gfCNCPoint5[6043] = {X 587.4990, Y 6.7049, Z -6.3333, A 0.000, B 0.000, C 0.000 }
gfCNCPoint5[6044] = {X 587.4271, Y 5.9692, Z -6.3333, A 0.000, B 0.000, C 0.000 }
gfCNCPoint5[6045] = {X 587.4270, Y 5.0000, Z -6.3333, A 0.000, B 0.000, C 0.000 }
gfCNCPoint5[6046] = {X 587.5313, Y 4.0743, Z -6.3333, A 0.000, B 0.000, C 0.000 }
gfCNCPoint5[6047] = {X 587.8389, Y 3.1950, Z -6.3333, A 0.000, B 0.000, C 0.000 }
gfCNCPoint5[6048] = {X 588.3345, Y 2.4063, Z -6.3333, A 0.000, B 0.000, C 0.000 }
gfCNCPoint5[6049] = {X 588.9932, Y 1.7476, Z -6.3333, A 0.000, B 0.000, C 0.000 }
gfCNCPoint5[6050] = {X 589.7820, Y 1.2520, Z -6.3333, A 0.000, B 0.000, C 0.000 }
gfCNCPoint5[6051] = {X 590.6613, Y 0.9443, Z -6.3333, A 0.000, B 0.000, C 0.000 }
gfCNCPoint5[6052] = {X 591.5870, Y 0.8400, Z -6.3333, A 0.000, B 0.000, C 0.000 }
gfCNCPoint5[6053] = {X 600.0000, Y 0.8400, Z -6.3333, A 0.000, B 0.000, C 0.000 }
gfCNCPoint5[6054] = {X 600.8245, Y 0.9225, Z -6.3333, A 0.000, B 0.000, C 0.000 }
gfCNCPoint5[6055] = {X 601.6162, Y 1.1668, Z -6.3333, A 0.000, B 0.000, C 0.000 }
gfCNCPoint5[6056] = {X 602.3439, Y 1.5632, Z -6.3333, A 0.000, B 0.000, C 0.000 }
gfCNCPoint5[6057] = {X 602.9785, Y 2.0959, Z -6.3333, A 0.000, B 0.000, C 0.000 }
gfCNCPoint5[6058] = {X 603.4950, Y 2.7438, Z -6.3333, A 0.000, B 0.000, C 0.000 }
gfCNCPoint5[6059] = {X 603.6000, Y 2.9154, Z -6.3333, A 0.000, B 0.000, C 0.000 }
gfCNCPoint5[6060] = {X 603.6966, Y 3.0920, Z -6.3333, A 0.000, B 0.000, C 0.000 }
gfCNCPoint5[6061] = {X 607.6966, Y 10.8417, Z -6.3333, A 0.000, B 0.000, C 0.000 }
gfCNCPoint5[6062] = {X 607.6966, Y 10.8417, Z -3.3333, A 0.000, B 0.000, C 0.000 }
gfCNCPoint5[6063] = {X 607.6966, Y 10.8417, Z 11.0000, A 0.000, B 0.000, C 0.000 }
gfCNCPoint5[6064] = {X 607.6966, Y 38.1629, Z 11.0000, A 0.000, B 0.000, C 0.000 }
gfCNCPoint5[6065] = {X 607.6966, Y 38.1629, Z -3.3333, A 0.000, B 0.000, C 0.000 }
gfCNCPoint5[6066] = {X 607.6966, Y 38.1629, Z -6.3333, A 0.000, B 0.000, C 0.000 }
gfCNCPoint5[6067] = {X 603.6966, Y 46.7266, Z -6.3333, A 0.000, B 0.000, C 0.000 }
gfCNCPoint5[6068] = {X 603.5705, Y 46.9743, Z -6.3333, A 0.000, B 0.000, C 0.000 }
gfCNCPoint5[6069] = {X 603.4278, Y 47.2128, Z -6.3333, A 0.000, B 0.000, C 0.000 }
gfCNCPoint5[6070] = {X 602.9212, Y 47.8483, Z -6.3333, A 0.000, B 0.000, C 0.000 }
gfCNCPoint5[6071] = {X 602.2988, Y 48.3708, Z -6.3333, A 0.000, B 0.000, C 0.000 }
gfCNCPoint5[6072] = {X 601.5851, Y 48.7595, Z -6.3333, A 0.000, B 0.000, C 0.000 }
gfCNCPoint5[6073] = {X 600.8086, Y 48.9991, Z -6.3333, A 0.000, B 0.000, C 0.000 }
gfCNCPoint5[6074] = {X 600.0000, Y 49.0800, Z -6.3333, A 0.000, B 0.000, C 0.000 }
gfCNCPoint5[6075] = {X 593.5565, Y 49.0800, Z -6.3333, A 0.000, B 0.000, C 0.000 }
gfCNCPoint5[6076] = {X 592.6486, Y 48.9777, Z -6.3333, A 0.000, B 0.000, C 0.000 }
gfCNCPoint5[6077] = {X 591.7863, Y 48.6760, Z -6.3333, A 0.000, B 0.000, C 0.000 }
gfCNCPoint5[6078] = {X 591.0127, Y 48.1899, Z -6.3333, A 0.000, B 0.000, C 0.000 }
gfCNCPoint5[6079] = {X 590.3667, Y 47.5438, Z -6.3333, A 0.000, B 0.000, C 0.000 }
gfCNCPoint5[6080] = {X 589.8806, Y 46.7702, Z -6.3333, A 0.000, B 0.000, C 0.000 }
gfCNCPoint5[6081] = {X 589.5788, Y 45.9079, Z -6.3333, A 0.000, B 0.000, C 0.000 }
gfCNCPoint5[6082] = {X 589.4765, Y 45.0000, Z -6.3333, A 0.000, B 0.000, C 0.000 }
gfCNCPoint5[6083] = {X 589.4765, Y 44.0656, Z -6.3333, A 0.000, B 0.000, C 0.000 }
gfCNCPoint5[6084] = {X 589.5808, Y 43.1618, Z -6.3333, A 0.000, B 0.000, C 0.000 }
gfCNCPoint5[6085] = {X 589.8809, Y 42.3029, Z -6.3333, A 0.000, B 0.000, C 0.000 }
gfCNCPoint5[6086] = {X 590.3624, Y 41.5308, Z -6.3333, A 0.000, B 0.000, C 0.000 }
gfCNCPoint5[6087] = {X 591.0016, Y 40.8833, Z -6.3333, A 0.000, B 0.000, C 0.000 }
gfCNCPoint5[6088] = {X 591.0024, Y 32.3007, Z -6.3333, A 0.000, B 0.000, C 0.000 }
gfCNCPoint5[6089] = {X 585.2236, Y 46.5606, Z -6.3333, A 0.000, B 0.000, C 0.000 }
gfCNCPoint5[6090] = {X 584.8743, Y 47.2242, Z -6.3333, A 0.000, B 0.000, C 0.000 }
gfCNCPoint5[6091] = {X 584.4095, Y 47.8125, Z -6.3333, A 0.000, B 0.000, C 0.000 }
gfCNCPoint5[6092] = {X 583.8449, Y 48.3059, Z -6.3333, A 0.000, B 0.000, C 0.000 }
gfCNCPoint5[6093] = {X 583.1996, Y 48.6877, Z -6.3333, A 0.000, B 0.000, C 0.000 }
gfCNCPoint5[6094] = {X 582.3082, Y 48.9895, Z -6.3333, A 0.000, B 0.000, C 0.000 }
gfCNCPoint5[6095] = {X 581.3715, Y 49.0792, Z -6.3333, A 0.000, B 0.000, C 0.000 }
gfCNCPoint5[6096] = {X 580.4391, Y 48.9518, Z -6.3333, A 0.000, B 0.000, C 0.000 }
gfCNCPoint5[6097] = {X 579.5607, Y 48.6142, Z -6.3333, A 0.000, B 0.000, C 0.000 }
gfCNCPoint5[6098] = {X 578.7830, Y 48.0843, Z -6.3333, A 0.000, B 0.000, C 0.000 }
gfCNCPoint5[6099] = {X 578.1474, Y 47.3903, Z -6.3333, A 0.000, B 0.000, C 0.000 }
gfCNCPoint5[6100] = {X 577.6877, Y 46.5692, Z -6.3333, A 0.000, B 0.000, C 0.000 }
gfCNCPoint5[6101] = {X 571.7795, Y 32.1221, Z -6.3333, A 0.000, B 0.000, C 0.000 }
gfCNCPoint5[6102] = {X 571.7798, Y 40.8840, Z -6.3333, A 0.000, B 0.000, C 0.000 }
gfCNCPoint5[6103] = {X 571.8686, Y 40.9570, Z -6.3333, A 0.000, B 0.000, C 0.000 }
gfCNCPoint5[6104] = {X 572.4697, Y 41.5905, Z -6.3333, A 0.000, B 0.000, C 0.000 }
gfCNCPoint5[6105] = {X 572.9222, Y 42.3373, Z -6.3333, A 0.000, B 0.000, C 0.000 }
gfCNCPoint5[6106] = {X 573.2054, Y 43.1634, Z -6.3333, A 0.000, B 0.000, C 0.000 }
gfCNCPoint5[6107] = {X 573.3063, Y 44.0308, Z -6.3333, A 0.000, B 0.000, C 0.000 }
gfCNCPoint5[6108] = {X 573.3064, Y 45.0000, Z -6.3333, A 0.000, B 0.000, C 0.000 }
gfCNCPoint5[6109] = {X 573.2041, Y 45.9079, Z -6.3333, A 0.000, B 0.000, C 0.000 }
gfCNCPoint5[6110] = {X 572.9024, Y 46.7702, Z -6.3333, A 0.000, B 0.000, C 0.000 }
gfCNCPoint5[6111] = {X 572.4163, Y 47.5438, Z -6.3333, A 0.000, B 0.000, C 0.000 }
gfCNCPoint5[6112] = {X 571.7703, Y 48.1899, Z -6.3333, A 0.000, B 0.000, C 0.000 }
gfCNCPoint5[6113] = {X 570.9967, Y 48.6760, Z -6.3333, A 0.000, B 0.000, C 0.000 }
gfCNCPoint5[6114] = {X 570.1343, Y 48.9777, Z -6.3333, A 0.000, B 0.000, C 0.000 }
gfCNCPoint5[6115] = {X 569.2264, Y 49.0800, Z -6.3333, A 0.000, B 0.000, C 0.000 }
gfCNCPoint5[6116] = {X 562.4443, Y 49.0800, Z -6.3333, A 0.000, B 0.000, C 0.000 }
gfCNCPoint5[6117] = {X 561.5364, Y 48.9777, Z -6.3333, A 0.000, B 0.000, C 0.000 }
gfCNCPoint5[6118] = {X 560.6741, Y 48.6760, Z -6.3333, A 0.000, B 0.000, C 0.000 }
gfCNCPoint5[6119] = {X 559.9005, Y 48.1899, Z -6.3333, A 0.000, B 0.000, C 0.000 }
gfCNCPoint5[6120] = {X 559.2544, Y 47.5438, Z -6.3333, A 0.000, B 0.000, C 0.000 }
gfCNCPoint5[6121] = {X 558.7683, Y 46.7702, Z -6.3333, A 0.000, B 0.000, C 0.000 }
gfCNCPoint5[6122] = {X 558.4666, Y 45.9079, Z -6.3333, A 0.000, B 0.000, C 0.000 }
gfCNCPoint5[6123] = {X 558.3643, Y 45.0000, Z -6.3333, A 0.000, B 0.000, C 0.000 }
gfCNCPoint5[6124] = {X 558.3643, Y 44.0657, Z -6.3333, A 0.000, B 0.000, C 0.000 }
gfCNCPoint5[6125] = {X 558.4683, Y 43.1614, Z -6.3333, A 0.000, B 0.000, C 0.000 }
gfCNCPoint5[6126] = {X 558.7688, Y 42.3022, Z -6.3333, A 0.000, B 0.000, C 0.000 }
gfCNCPoint5[6127] = {X 559.2510, Y 41.5302, Z -6.3333, A 0.000, B 0.000, C 0.000 }
gfCNCPoint5[6128] = {X 559.8912, Y 40.8832, Z -6.3333, A 0.000, B 0.000, C 0.000 }
gfCNCPoint5[6129] = {X 559.8912, Y 9.1165, Z -6.3333, A 0.000, B 0.000, C 0.000 }
gfCNCPoint5[6130] = {X 559.2544, Y 8.4779, Z -6.3333, A 0.000, B 0.000, C 0.000 }
gfCNCPoint5[6131] = {X 558.7735, Y 7.7150, Z -6.3333, A 0.000, B 0.000, C 0.000 }
gfCNCPoint5[6132] = {X 558.4720, Y 6.8651, Z -6.3333, A 0.000, B 0.000, C 0.000 }
gfCNCPoint5[6133] = {X 558.3645, Y 5.9697, Z -6.3333, A 0.000, B 0.000, C 0.000 }
gfCNCPoint5[6134] = {X 558.3643, Y 5.0000, Z -6.3333, A 0.000, B 0.000, C 0.000 }
gfCNCPoint5[6135] = {X 558.4666, Y 4.0921, Z -6.3333, A 0.000, B 0.000, C 0.000 }
gfCNCPoint5[6136] = {X 558.7683, Y 3.2298, Z -6.3333, A 0.000, B 0.000, C 0.000 }
gfCNCPoint5[6137] = {X 559.2544, Y 2.4562, Z -6.3333, A 0.000, B 0.000, C 0.000 }
gfCNCPoint5[6138] = {X 559.9005, Y 1.8101, Z -6.3333, A 0.000, B 0.000, C 0.000 }
gfCNCPoint5[6139] = {X 560.6741, Y 1.3240, Z -6.3333, A 0.000, B 0.000, C 0.000 }
gfCNCPoint5[6140] = {X 561.5364, Y 1.0223, Z -6.3333, A 0.000, B 0.000, C 0.000 }
gfCNCPoint5[6141] = {X 562.4443, Y 0.9200, Z -6.3333, A 0.000, B 0.000, C 0.000 }
gfCNCPoint5[6142] = {X 570.9376, Y 0.9200, Z -6.3333, A 0.000, B 0.000, C 0.000 }
gfCNCPoint5[6143] = {X 571.8454, Y 1.0223, Z -6.3333, A 0.000, B 0.000, C 0.000 }
gfCNCPoint5[6144] = {X 572.7078, Y 1.3240, Z -6.3333, A 0.000, B 0.000, C 0.000 }
gfCNCPoint5[6145] = {X 573.4814, Y 1.8101, Z -6.3333, A 0.000, B 0.000, C 0.000 }
gfCNCPoint5[6146] = {X 574.1274, Y 2.4562, Z -6.3333, A 0.000, B 0.000, C 0.000 }
gfCNCPoint5[6147] = {X 574.6135, Y 3.2298, Z -6.3333, A 0.000, B 0.000, C 0.000 }
gfCNCPoint5[6148] = {X 574.9153, Y 4.0921, Z -6.3333, A 0.000, B 0.000, C 0.000 }
gfCNCPoint5[6149] = {X 575.0176, Y 5.0000, Z -6.3333, A 0.000, B 0.000, C 0.000 }
gfCNCPoint5[6150] = {X 575.0176, Y 5.9342, Z -6.3333, A 0.000, B 0.000, C 0.000 }
gfCNCPoint5[6151] = {X 574.9500, Y 6.6733, Z -6.3333, A 0.000, B 0.000, C 0.000 }
gfCNCPoint5[6152] = {X 574.7497, Y 7.3880, Z -6.3333, A 0.000, B 0.000, C 0.000 }
gfCNCPoint5[6153] = {X 574.4233, Y 8.0545, Z -6.3333, A 0.000, B 0.000, C 0.000 }
gfCNCPoint5[6154] = {X 574.3788, Y 8.1258, Z -6.3333, A 0.000, B 0.000, C 0.000 }
gfCNCPoint5[6155] = {X 574.3330, Y 8.1963, Z -6.3333, A 0.000, B 0.000, C 0.000 }
gfCNCPoint5[6156] = {X 574.3593, Y 8.2418, Z -6.3333, A 0.000, B 0.000, C 0.000 }
gfCNCPoint5[6157] = {X 581.1906, Y 25.0042, Z -6.3333, A 0.000, B 0.000, C 0.000 }
gfCNCPoint5[6158] = {X 588.1131, Y 8.0738, Z -6.3333, A 0.000, B 0.000, C 0.000 }
gfCNCPoint5[6159] = {X 587.7843, Y 7.4127, Z -6.3333, A 0.000, B 0.000, C 0.000 }
gfCNCPoint5[6160] = {X 587.5801, Y 6.7032, Z -6.3333, A 0.000, B 0.000, C 0.000 }
gfCNCPoint5[6161] = {X 587.5071, Y 5.9685, Z -6.3333, A 0.000, B 0.000, C 0.000 }
gfCNCPoint5[6162] = {X 587.5070, Y 5.0000, Z -6.3333, A 0.000, B 0.000, C 0.000 }
gfCNCPoint5[6163] = {X 587.6092, Y 4.0921, Z -6.3333, A 0.000, B 0.000, C 0.000 }
gfCNCPoint5[6164] = {X 587.9110, Y 3.2298, Z -6.3333, A 0.000, B 0.000, C 0.000 }
gfCNCPoint5[6165] = {X 588.3971, Y 2.4562, Z -6.3333, A 0.000, B 0.000, C 0.000 }
gfCNCPoint5[6166] = {X 589.0431, Y 1.8101, Z -6.3333, A 0.000, B 0.000, C 0.000 }
gfCNCPoint5[6167] = {X 589.8167, Y 1.3240, Z -6.3333, A 0.000, B 0.000, C 0.000 }
gfCNCPoint5[6168] = {X 590.6791, Y 1.0223, Z -6.3333, A 0.000, B 0.000, C 0.000 }
gfCNCPoint5[6169] = {X 591.5870, Y 0.9200, Z -6.3333, A 0.000, B 0.000, C 0.000 }
gfCNCPoint5[6170] = {X 600.0000, Y 0.9200, Z -6.3333, A 0.000, B 0.000, C 0.000 }
gfCNCPoint5[6171] = {X 600.8086, Y 1.0009, Z -6.3333, A 0.000, B 0.000, C 0.000 }
gfCNCPoint5[6172] = {X 601.5851, Y 1.2405, Z -6.3333, A 0.000, B 0.000, C 0.000 }
gfCNCPoint5[6173] = {X 602.2988, Y 1.6292, Z -6.3333, A 0.000, B 0.000, C 0.000 }
gfCNCPoint5[6174] = {X 602.9212, Y 2.1517, Z -6.3333, A 0.000, B 0.000, C 0.000 }
gfCNCPoint5[6175] = {X 603.4278, Y 2.7872, Z -6.3333, A 0.000, B 0.000, C 0.000 }
gfCNCPoint5[6176] = {X 603.5705, Y 3.0257, Z -6.3333, A 0.000, B 0.000, C 0.000 }
gfCNCPoint5[6177] = {X 603.6966, Y 3.2734, Z -6.3333, A 0.000, B 0.000, C 0.000 }
gfCNCPoint5[6178] = {X 607.6966, Y 11.8371, Z -6.3333, A 0.000, B 0.000, C 0.000 }
gfCNCPoint5[6179] = {X 607.6966, Y 11.8371, Z -3.3333, A 0.000, B 0.000, C 0.000 }
gfCNCPoint5[6180] = {X 607.6966, Y 11.8371, Z 11.0000, A 0.000, B 0.000, C 0.000 }
gfCNCPoint5[6181] = {X 607.6966, Y 36.8512, Z 11.0000, A 0.000, B 0.000, C 0.000 }
gfCNCPoint5[6182] = {X 607.6966, Y 36.8512, Z -3.3333, A 0.000, B 0.000, C 0.000 }
gfCNCPoint5[6183] = {X 607.6966, Y 36.8512, Z -6.3333, A 0.000, B 0.000, C 0.000 }
gfCNCPoint5[6184] = {X 603.6966, Y 46.5280, Z -6.3333, A 0.000, B 0.000, C 0.000 }
gfCNCPoint5[6185] = {X 603.5432, Y 46.8564, Z -6.3333, A 0.000, B 0.000, C 0.000 }
gfCNCPoint5[6186] = {X 603.3606, Y 47.1694, Z -6.3333, A 0.000, B 0.000, C 0.000 }
gfCNCPoint5[6187] = {X 602.8640, Y 47.7924, Z -6.3333, A 0.000, B 0.000, C 0.000 }
gfCNCPoint5[6188] = {X 602.2537, Y 48.3047, Z -6.3333, A 0.000, B 0.000, C 0.000 }
gfCNCPoint5[6189] = {X 601.5541, Y 48.6858, Z -6.3333, A 0.000, B 0.000, C 0.000 }
gfCNCPoint5[6190] = {X 600.7928, Y 48.9207, Z -6.3333, A 0.000, B 0.000, C 0.000 }
gfCNCPoint5[6191] = {X 600.0000, Y 49.0000, Z -6.3333, A 0.000, B 0.000, C 0.000 }
gfCNCPoint5[6192] = {X 593.5565, Y 49.0000, Z -6.3333, A 0.000, B 0.000, C 0.000 }
gfCNCPoint5[6193] = {X 592.6664, Y 48.8997, Z -6.3333, A 0.000, B 0.000, C 0.000 }
gfCNCPoint5[6194] = {X 591.8210, Y 48.6039, Z -6.3333, A 0.000, B 0.000, C 0.000 }
gfCNCPoint5[6195] = {X 591.0626, Y 48.1273, Z -6.3333, A 0.000, B 0.000, C 0.000 }
gfCNCPoint5[6196] = {X 590.4292, Y 47.4940, Z -6.3333, A 0.000, B 0.000, C 0.000 }
gfCNCPoint5[6197] = {X 589.9527, Y 46.7355, Z -6.3333, A 0.000, B 0.000, C 0.000 }
gfCNCPoint5[6198] = {X 589.6568, Y 45.8901, Z -6.3333, A 0.000, B 0.000, C 0.000 }
gfCNCPoint5[6199] = {X 589.5565, Y 45.0000, Z -6.3333, A 0.000, B 0.000, C 0.000 }
gfCNCPoint5[6200] = {X 589.5565, Y 44.0660, Z -6.3333, A 0.000, B 0.000, C 0.000 }
gfCNCPoint5[6201] = {X 589.6609, Y 43.1705, Z -6.3333, A 0.000, B 0.000, C 0.000 }
gfCNCPoint5[6202] = {X 589.9613, Y 42.3204, Z -6.3333, A 0.000, B 0.000, C 0.000 }
gfCNCPoint5[6203] = {X 590.4428, Y 41.5582, Z -6.3333, A 0.000, B 0.000, C 0.000 }
gfCNCPoint5[6204] = {X 591.0815, Y 40.9218, Z -6.3333, A 0.000, B 0.000, C 0.000 }
gfCNCPoint5[6205] = {X 591.0821, Y 40.7351, Z -6.3333, A 0.000, B 0.000, C 0.000 }
gfCNCPoint5[6206] = {X 591.0834, Y 40.3069, Z -6.3333, A 0.000, B 0.000, C 0.000 }
gfCNCPoint5[6207] = {X 591.0823, Y 32.0438, Z -6.3333, A 0.000, B 0.000, C 0.000 }
gfCNCPoint5[6208] = {X 590.9675, Y 32.1736, Z -6.3333, A 0.000, B 0.000, C 0.000 }
gfCNCPoint5[6209] = {X 590.3119, Y 33.7916, Z -6.3333, A 0.000, B 0.000, C 0.000 }
gfCNCPoint5[6210] = {X 585.1497, Y 46.5300, Z -6.3333, A 0.000, B 0.000, C 0.000 }
gfCNCPoint5[6211] = {X 584.8073, Y 47.1805, Z -6.3333, A 0.000, B 0.000, C 0.000 }
gfCNCPoint5[6212] = {X 584.3516, Y 47.7574, Z -6.3333, A 0.000, B 0.000, C 0.000 }
gfCNCPoint5[6213] = {X 583.7980, Y 48.2411, Z -6.3333, A 0.000, B 0.000, C 0.000 }
gfCNCPoint5[6214] = {X 583.1653, Y 48.6154, Z -6.3333, A 0.000, B 0.000, C 0.000 }
gfCNCPoint5[6215] = {X 582.2878, Y 48.9121, Z -6.3333, A 0.000, B 0.000, C 0.000 }
gfCNCPoint5[6216] = {X 581.3656, Y 48.9990, Z -6.3333, A 0.000, B 0.000, C 0.000 }
gfCNCPoint5[6217] = {X 580.4480, Y 48.8715, Z -6.3333, A 0.000, B 0.000, C 0.000 }
gfCNCPoint5[6218] = {X 579.5845, Y 48.5363, Z -6.3333, A 0.000, B 0.000, C 0.000 }
gfCNCPoint5[6219] = {X 578.8212, Y 48.0115, Z -6.3333, A 0.000, B 0.000, C 0.000 }
gfCNCPoint5[6220] = {X 578.1990, Y 47.3251, Z -6.3333, A 0.000, B 0.000, C 0.000 }
gfCNCPoint5[6221] = {X 577.7515, Y 46.5141, Z -6.3333, A 0.000, B 0.000, C 0.000 }
gfCNCPoint5[6222] = {X 571.6995, Y 31.7151, Z -6.3333, A 0.000, B 0.000, C 0.000 }
gfCNCPoint5[6223] = {X 571.6998, Y 40.9218, Z -6.3333, A 0.000, B 0.000, C 0.000 }
gfCNCPoint5[6224] = {X 571.8386, Y 41.0366, Z -6.3333, A 0.000, B 0.000, C 0.000 }
gfCNCPoint5[6225] = {X 572.4243, Y 41.6631, Z -6.3333, A 0.000, B 0.000, C 0.000 }
gfCNCPoint5[6226] = {X 572.8630, Y 42.3999, Z -6.3333, A 0.000, B 0.000, C 0.000 }
gfCNCPoint5[6227] = {X 573.1345, Y 43.2134, Z -6.3333, A 0.000, B 0.000, C 0.000 }
gfCNCPoint5[6228] = {X 573.2264, Y 44.0660, Z -6.3333, A 0.000, B 0.000, C 0.000 }
gfCNCPoint5[6229] = {X 573.2264, Y 45.0000, Z -6.3333, A 0.000, B 0.000, C 0.000 }
gfCNCPoint5[6230] = {X 573.1261, Y 45.8901, Z -6.3333, A 0.000, B 0.000, C 0.000 }
gfCNCPoint5[6231] = {X 572.8303, Y 46.7355, Z -6.3333, A 0.000, B 0.000, C 0.000 }
gfCNCPoint5[6232] = {X 572.3538, Y 47.4940, Z -6.3333, A 0.000, B 0.000, C 0.000 }
gfCNCPoint5[6233] = {X 571.7204, Y 48.1273, Z -6.3333, A 0.000, B 0.000, C 0.000 }
gfCNCPoint5[6234] = {X 570.9620, Y 48.6039, Z -6.3333, A 0.000, B 0.000, C 0.000 }
gfCNCPoint5[6235] = {X 570.1165, Y 48.8997, Z -6.3333, A 0.000, B 0.000, C 0.000 }
gfCNCPoint5[6236] = {X 569.2264, Y 49.0000, Z -6.3333, A 0.000, B 0.000, C 0.000 }
gfCNCPoint5[6237] = {X 562.4443, Y 49.0000, Z -6.3333, A 0.000, B 0.000, C 0.000 }
gfCNCPoint5[6238] = {X 561.5542, Y 48.8997, Z -6.3333, A 0.000, B 0.000, C 0.000 }
gfCNCPoint5[6239] = {X 560.7088, Y 48.6039, Z -6.3333, A 0.000, B 0.000, C 0.000 }
gfCNCPoint5[6240] = {X 559.9503, Y 48.1273, Z -6.3333, A 0.000, B 0.000, C 0.000 }
gfCNCPoint5[6241] = {X 559.3170, Y 47.4940, Z -6.3333, A 0.000, B 0.000, C 0.000 }
gfCNCPoint5[6242] = {X 558.8404, Y 46.7355, Z -6.3333, A 0.000, B 0.000, C 0.000 }
gfCNCPoint5[6243] = {X 558.5446, Y 45.8901, Z -6.3333, A 0.000, B 0.000, C 0.000 }
gfCNCPoint5[6244] = {X 558.4443, Y 45.0000, Z -6.3333, A 0.000, B 0.000, C 0.000 }
gfCNCPoint5[6245] = {X 558.4443, Y 44.0660, Z -6.3333, A 0.000, B 0.000, C 0.000 }
gfCNCPoint5[6246] = {X 558.5484, Y 43.1700, Z -6.3333, A 0.000, B 0.000, C 0.000 }
gfCNCPoint5[6247] = {X 558.8492, Y 42.3197, Z -6.3333, A 0.000, B 0.000, C 0.000 }
gfCNCPoint5[6248] = {X 559.3315, Y 41.5575, Z -6.3333, A 0.000, B 0.000, C 0.000 }
gfCNCPoint5[6249] = {X 559.9712, Y 40.9217, Z -6.3333, A 0.000, B 0.000, C 0.000 }
gfCNCPoint5[6250] = {X 559.9712, Y 9.0779, Z -6.3333, A 0.000, B 0.000, C 0.000 }
gfCNCPoint5[6251] = {X 559.3294, Y 8.4436, Z -6.3333, A 0.000, B 0.000, C 0.000 }
gfCNCPoint5[6252] = {X 558.8462, Y 7.6815, Z -6.3333, A 0.000, B 0.000, C 0.000 }
gfCNCPoint5[6253] = {X 558.5461, Y 6.8306, Z -6.3333, A 0.000, B 0.000, C 0.000 }
gfCNCPoint5[6254] = {X 558.4443, Y 5.9340, Z -6.3333, A 0.000, B 0.000, C 0.000 }
gfCNCPoint5[6255] = {X 558.4443, Y 5.0000, Z -6.3333, A 0.000, B 0.000, C 0.000 }
gfCNCPoint5[6256] = {X 558.5446, Y 4.1099, Z -6.3333, A 0.000, B 0.000, C 0.000 }
gfCNCPoint5[6257] = {X 558.8404, Y 3.2645, Z -6.3333, A 0.000, B 0.000, C 0.000 }
gfCNCPoint5[6258] = {X 559.3170, Y 2.5060, Z -6.3333, A 0.000, B 0.000, C 0.000 }
gfCNCPoint5[6259] = {X 559.9503, Y 1.8727, Z -6.3333, A 0.000, B 0.000, C 0.000 }
gfCNCPoint5[6260] = {X 560.7088, Y 1.3961, Z -6.3333, A 0.000, B 0.000, C 0.000 }
gfCNCPoint5[6261] = {X 561.5542, Y 1.1003, Z -6.3333, A 0.000, B 0.000, C 0.000 }
gfCNCPoint5[6262] = {X 562.4443, Y 1.0000, Z -6.3333, A 0.000, B 0.000, C 0.000 }
gfCNCPoint5[6263] = {X 570.9376, Y 1.0000, Z -6.3333, A 0.000, B 0.000, C 0.000 }
gfCNCPoint5[6264] = {X 571.8276, Y 1.1003, Z -6.3333, A 0.000, B 0.000, C 0.000 }
gfCNCPoint5[6265] = {X 572.6731, Y 1.3961, Z -6.3333, A 0.000, B 0.000, C 0.000 }
gfCNCPoint5[6266] = {X 573.4315, Y 1.8727, Z -6.3333, A 0.000, B 0.000, C 0.000 }
gfCNCPoint5[6267] = {X 574.0649, Y 2.5060, Z -6.3333, A 0.000, B 0.000, C 0.000 }
gfCNCPoint5[6268] = {X 574.5414, Y 3.2645, Z -6.3333, A 0.000, B 0.000, C 0.000 }
gfCNCPoint5[6269] = {X 574.8373, Y 4.1099, Z -6.3333, A 0.000, B 0.000, C 0.000 }
gfCNCPoint5[6270] = {X 574.9376, Y 5.0000, Z -6.3333, A 0.000, B 0.000, C 0.000 }
gfCNCPoint5[6271] = {X 574.9372, Y 5.9858, Z -6.3333, A 0.000, B 0.000, C 0.000 }
gfCNCPoint5[6272] = {X 574.8650, Y 6.6926, Z -6.3333, A 0.000, B 0.000, C 0.000 }
gfCNCPoint5[6273] = {X 574.6688, Y 7.3755, Z -6.3333, A 0.000, B 0.000, C 0.000 }
gfCNCPoint5[6274] = {X 574.3549, Y 8.0129, Z -6.3333, A 0.000, B 0.000, C 0.000 }
gfCNCPoint5[6275] = {X 574.2921, Y 8.1128, Z -6.3333, A 0.000, B 0.000, C 0.000 }
gfCNCPoint5[6276] = {X 574.2264, Y 8.2108, Z -6.3333, A 0.000, B 0.000, C 0.000 }
gfCNCPoint5[6277] = {X 574.2617, Y 8.2359, Z -6.3333, A 0.000, B 0.000, C 0.000 }
gfCNCPoint5[6278] = {X 574.2853, Y 8.2722, Z -6.3333, A 0.000, B 0.000, C 0.000 }
gfCNCPoint5[6279] = {X 574.9161, Y 9.8071, Z -6.3333, A 0.000, B 0.000, C 0.000 }
gfCNCPoint5[6280] = {X 581.1904, Y 25.2159, Z -6.3333, A 0.000, B 0.000, C 0.000 }
gfCNCPoint5[6281] = {X 588.2026, Y 8.0662, Z -6.3333, A 0.000, B 0.000, C 0.000 }
gfCNCPoint5[6282] = {X 587.8646, Y 7.3984, Z -6.3333, A 0.000, B 0.000, C 0.000 }
gfCNCPoint5[6283] = {X 587.6570, Y 6.6792, Z -6.3333, A 0.000, B 0.000, C 0.000 }
gfCNCPoint5[6284] = {X 587.5870, Y 5.9340, Z -6.3333, A 0.000, B 0.000, C 0.000 }
gfCNCPoint5[6285] = {X 587.5870, Y 5.0000, Z -6.3333, A 0.000, B 0.000, C 0.000 }
gfCNCPoint5[6286] = {X 587.6872, Y 4.1099, Z -6.3333, A 0.000, B 0.000, C 0.000 }
gfCNCPoint5[6287] = {X 587.9831, Y 3.2645, Z -6.3333, A 0.000, B 0.000, C 0.000 }
gfCNCPoint5[6288] = {X 588.4596, Y 2.5060, Z -6.3333, A 0.000, B 0.000, C 0.000 }
gfCNCPoint5[6289] = {X 589.0930, Y 1.8727, Z -6.3333, A 0.000, B 0.000, C 0.000 }
gfCNCPoint5[6290] = {X 589.8514, Y 1.3961, Z -6.3333, A 0.000, B 0.000, C 0.000 }
gfCNCPoint5[6291] = {X 590.6969, Y 1.1003, Z -6.3333, A 0.000, B 0.000, C 0.000 }
gfCNCPoint5[6292] = {X 591.5870, Y 1.0000, Z -6.3333, A 0.000, B 0.000, C 0.000 }
gfCNCPoint5[6293] = {X 600.0000, Y 1.0000, Z -6.3333, A 0.000, B 0.000, C 0.000 }
gfCNCPoint5[6294] = {X 600.7928, Y 1.0793, Z -6.3333, A 0.000, B 0.000, C 0.000 }
gfCNCPoint5[6295] = {X 601.5541, Y 1.3142, Z -6.3333, A 0.000, B 0.000, C 0.000 }
gfCNCPoint5[6296] = {X 602.2537, Y 1.6953, Z -6.3333, A 0.000, B 0.000, C 0.000 }
gfCNCPoint5[6297] = {X 602.8640, Y 2.2076, Z -6.3333, A 0.000, B 0.000, C 0.000 }
gfCNCPoint5[6298] = {X 603.3606, Y 2.8306, Z -6.3333, A 0.000, B 0.000, C 0.000 }
gfCNCPoint5[6299] = {X 603.5432, Y 3.1436, Z -6.3333, A 0.000, B 0.000, C 0.000 }
gfCNCPoint5[6300] = {X 603.6966, Y 3.4720, Z -6.3333, A 0.000, B 0.000, C 0.000 }
gfCNCPoint5[6301] = {X 607.6966, Y 13.1488, Z -6.3333, A 0.000, B 0.000, C 0.000 }
gfCNCPoint5[6302] = {X 607.6966, Y 13.1488, Z -3.3333, A 0.000, B 0.000, C 0.000 }
gfCNCPoint5[6303] = {X 607.6966, Y 13.1488, Z 11.0000, A 0.000, B 0.000, C 0.000 }
gfCNCPoint5[6304] = {X 256.2463, Y 19.7817, Z 11.0000, A 0.000, B 0.000, C 0.000 }
gfCNCPoint5[6305] = {X 256.2463, Y 19.7817, Z -2.5000, A 0.000, B 0.000, C 0.000 }
gfCNCPoint5[6306] = {X 251.5292, Y 19.7817, Z -3.7639, A 0.000, B 0.000, C 0.000 }
gfCNCPoint5[6307] = {X 250.8344, Y 19.7926, Z -3.9501, A 0.000, B 0.000, C 0.000 }
gfCNCPoint5[6308] = {X 250.1815, Y 19.7939, Z -4.1251, A 0.000, B 0.000, C 0.000 }
gfCNCPoint5[6309] = {X 249.4949, Y 19.8924, Z -4.3110, A 0.000, B 0.000, C 0.000 }
gfCNCPoint5[6310] = {X 248.8454, Y 20.0807, Z -4.4922, A 0.000, B 0.000, C 0.000 }
gfCNCPoint5[6311] = {X 248.7086, Y 20.1119, Z -4.5298, A 0.000, B 0.000, C 0.000 }
gfCNCPoint5[6312] = {X 248.6548, Y 20.1623, Z -4.5495, A 0.000, B 0.000, C 0.000 }
gfCNCPoint5[6313] = {X 248.6149, Y 20.2969, Z -4.5871, A 0.000, B 0.000, C 0.000 }
gfCNCPoint5[6314] = {X 248.4759, Y 20.7652, Z -4.7180, A 0.000, B 0.000, C 0.000 }
gfCNCPoint5[6315] = {X 248.4457, Y 21.8668, Z -5.0133, A 0.000, B 0.000, C 0.000 }
gfCNCPoint5[6316] = {X 248.5589, Y 22.3420, Z -5.1442, A 0.000, B 0.000, C 0.000 }
gfCNCPoint5[6317] = {X 248.8757, Y 22.4372, Z -5.2328, A 0.000, B 0.000, C 0.000 }
gfCNCPoint5[6318] = {X 250.4427, Y 22.5655, Z -5.6541, A 0.000, B 0.000, C 0.000 }
gfCNCPoint5[6319] = {X 251.6873, Y 22.5560, Z -5.9876, A 0.000, B 0.000, C 0.000 }
gfCNCPoint5[6320] = {X 252.9776, Y 22.5560, Z -6.3333, A 0.000, B 0.000, C 0.000 }
gfCNCPoint5[6321] = {X 257.4115, Y 22.5560, Z -6.3333, A 0.000, B 0.000, C 0.000 }
gfCNCPoint5[6322] = {X 257.4115, Y 19.7817, Z -6.3333, A 0.000, B 0.000, C 0.000 }
gfCNCPoint5[6323] = {X 251.5292, Y 19.7817, Z -6.3333, A 0.000, B 0.000, C 0.000 }
gfCNCPoint5[6324] = {X 250.8344, Y 19.7926, Z -6.3333, A 0.000, B 0.000, C 0.000 }
gfCNCPoint5[6325] = {X 249.8296, Y 19.8658, Z -6.3333, A 0.000, B 0.000, C 0.000 }
gfCNCPoint5[6326] = {X 248.8454, Y 20.0807, Z -6.3333, A 0.000, B 0.000, C 0.000 }
gfCNCPoint5[6327] = {X 248.7009, Y 20.1576, Z -6.3333, A 0.000, B 0.000, C 0.000 }
gfCNCPoint5[6328] = {X 248.6149, Y 20.2969, Z -6.3333, A 0.000, B 0.000, C 0.000 }
gfCNCPoint5[6329] = {X 248.4770, Y 20.9719, Z -6.3333, A 0.000, B 0.000, C 0.000 }
gfCNCPoint5[6330] = {X 248.4582, Y 21.6605, Z -6.3333, A 0.000, B 0.000, C 0.000 }
gfCNCPoint5[6331] = {X 248.5589, Y 22.3420, Z -6.3333, A 0.000, B 0.000, C 0.000 }
gfCNCPoint5[6332] = {X 248.8789, Y 22.4201, Z -6.3333, A 0.000, B 0.000, C 0.000 }
gfCNCPoint5[6333] = {X 249.2053, Y 22.4642, Z -6.3333, A 0.000, B 0.000, C 0.000 }
gfCNCPoint5[6334] = {X 250.4453, Y 22.5379, Z -6.3333, A 0.000, B 0.000, C 0.000 }
gfCNCPoint5[6335] = {X 251.6873, Y 22.5560, Z -6.3333, A 0.000, B 0.000, C 0.000 }
gfCNCPoint5[6336] = {X 252.9776, Y 22.5560, Z -6.3333, A 0.000, B 0.000, C 0.000 }
gfCNCPoint5[6337] = {X 248.9928, Y 22.2874, Z -6.3333, A 0.000, B 0.000, C 0.000 }
gfCNCPoint5[6338] = {X 252.9776, Y 22.6360, Z -6.3333, A 0.000, B 0.000, C 0.000 }
gfCNCPoint5[6339] = {X 257.4915, Y 22.6360, Z -6.3333, A 0.000, B 0.000, C 0.000 }
gfCNCPoint5[6340] = {X 257.4915, Y 19.7017, Z -6.3333, A 0.000, B 0.000, C 0.000 }
gfCNCPoint5[6341] = {X 251.5286, Y 19.7017, Z -6.3333, A 0.000, B 0.000, C 0.000 }
gfCNCPoint5[6342] = {X 250.8364, Y 19.7126, Z -6.3333, A 0.000, B 0.000, C 0.000 }
gfCNCPoint5[6343] = {X 249.8259, Y 19.7859, Z -6.3333, A 0.000, B 0.000, C 0.000 }
gfCNCPoint5[6344] = {X 248.8357, Y 20.0009, Z -6.3333, A 0.000, B 0.000, C 0.000 }
gfCNCPoint5[6345] = {X 248.6492, Y 20.0964, Z -6.3333, A 0.000, B 0.000, C 0.000 }
gfCNCPoint5[6346] = {X 248.5382, Y 20.2741, Z -6.3333, A 0.000, B 0.000, C 0.000 }
gfCNCPoint5[6347] = {X 248.3958, Y 20.9779, Z -6.3333, A 0.000, B 0.000, C 0.000 }
gfCNCPoint5[6348] = {X 248.3803, Y 21.6958, Z -6.3333, A 0.000, B 0.000, C 0.000 }
gfCNCPoint5[6349] = {X 248.4919, Y 22.4051, Z -6.3333, A 0.000, B 0.000, C 0.000 }
gfCNCPoint5[6350] = {X 248.8415, Y 22.4943, Z -6.3333, A 0.000, B 0.000, C 0.000 }
gfCNCPoint5[6351] = {X 249.1988, Y 22.5439, Z -6.3333, A 0.000, B 0.000, C 0.000 }
gfCNCPoint5[6352] = {X 250.4414, Y 22.6178, Z -6.3333, A 0.000, B 0.000, C 0.000 }
gfCNCPoint5[6353] = {X 251.6861, Y 22.6360, Z -6.3333, A 0.000, B 0.000, C 0.000 }
gfCNCPoint5[6354] = {X 252.9776, Y 22.6360, Z -6.3333, A 0.000, B 0.000, C 0.000 }
gfCNCPoint5[6355] = {X 256.9624, Y 22.2874, Z -6.3333, A 0.000, B 0.000, C 0.000 }
gfCNCPoint5[6356] = {X 248.9928, Y 22.3674, Z -6.3333, A 0.000, B 0.000, C 0.000 }
gfCNCPoint5[6357] = {X 252.9776, Y 22.7160, Z -6.3333, A 0.000, B 0.000, C 0.000 }
gfCNCPoint5[6358] = {X 257.5715, Y 22.7160, Z -6.3333, A 0.000, B 0.000, C 0.000 }
gfCNCPoint5[6359] = {X 257.5715, Y 19.6217, Z -6.3333, A 0.000, B 0.000, C 0.000 }
gfCNCPoint5[6360] = {X 251.5280, Y 19.6217, Z -6.3333, A 0.000, B 0.000, C 0.000 }
gfCNCPoint5[6361] = {X 250.8357, Y 19.6326, Z -6.3333, A 0.000, B 0.000, C 0.000 }
gfCNCPoint5[6362] = {X 249.8156, Y 19.7065, Z -6.3333, A 0.000, B 0.000, C 0.000 }
gfCNCPoint5[6363] = {X 248.8161, Y 19.9232, Z -6.3333, A 0.000, B 0.000, C 0.000 }
gfCNCPoint5[6364] = {X 248.5938, Y 20.0386, Z -6.3333, A 0.000, B 0.000, C 0.000 }
gfCNCPoint5[6365] = {X 248.4615, Y 20.2513, Z -6.3333, A 0.000, B 0.000, C 0.000 }
gfCNCPoint5[6366] = {X 248.3147, Y 20.9838, Z -6.3333, A 0.000, B 0.000, C 0.000 }
gfCNCPoint5[6367] = {X 248.3025, Y 21.7308, Z -6.3333, A 0.000, B 0.000, C 0.000 }
gfCNCPoint5[6368] = {X 248.4254, Y 22.4676, Z -6.3333, A 0.000, B 0.000, C 0.000 }
gfCNCPoint5[6369] = {X 248.8042, Y 22.5685, Z -6.3333, A 0.000, B 0.000, C 0.000 }
gfCNCPoint5[6370] = {X 249.1923, Y 22.6236, Z -6.3333, A 0.000, B 0.000, C 0.000 }
gfCNCPoint5[6371] = {X 250.4383, Y 22.6977, Z -6.3333, A 0.000, B 0.000, C 0.000 }
gfCNCPoint5[6372] = {X 251.6864, Y 22.7160, Z -6.3333, A 0.000, B 0.000, C 0.000 }
gfCNCPoint5[6373] = {X 252.9776, Y 22.7160, Z -6.3333, A 0.000, B 0.000, C 0.000 }
gfCNCPoint5[6374] = {X 256.9624, Y 22.3674, Z -6.3333, A 0.000, B 0.000, C 0.000 }
gfCNCPoint5[6375] = {X 248.9928, Y 22.4474, Z -6.3333, A 0.000, B 0.000, C 0.000 }
gfCNCPoint5[6376] = {X 252.9776, Y 22.7960, Z -6.3333, A 0.000, B 0.000, C 0.000 }
gfCNCPoint5[6377] = {X 257.6515, Y 22.7960, Z -6.3333, A 0.000, B 0.000, C 0.000 }
gfCNCPoint5[6378] = {X 257.6515, Y 19.5417, Z -6.3333, A 0.000, B 0.000, C 0.000 }
gfCNCPoint5[6379] = {X 251.5274, Y 19.5417, Z -6.3333, A 0.000, B 0.000, C 0.000 }
gfCNCPoint5[6380] = {X 250.8350, Y 19.5526, Z -6.3333, A 0.000, B 0.000, C 0.000 }
gfCNCPoint5[6381] = {X 249.8053, Y 19.6272, Z -6.3333, A 0.000, B 0.000, C 0.000 }
gfCNCPoint5[6382] = {X 248.7963, Y 19.8457, Z -6.3333, A 0.000, B 0.000, C 0.000 }
gfCNCPoint5[6383] = {X 248.5383, Y 19.9810, Z -6.3333, A 0.000, B 0.000, C 0.000 }
gfCNCPoint5[6384] = {X 248.3848, Y 20.2286, Z -6.3333, A 0.000, B 0.000, C 0.000 }
gfCNCPoint5[6385] = {X 248.2337, Y 20.9896, Z -6.3333, A 0.000, B 0.000, C 0.000 }
gfCNCPoint5[6386] = {X 248.2250, Y 21.7655, Z -6.3333, A 0.000, B 0.000, C 0.000 }
gfCNCPoint5[6387] = {X 248.3592, Y 22.5297, Z -6.3333, A 0.000, B 0.000, C 0.000 }
gfCNCPoint5[6388] = {X 248.7670, Y 22.6425, Z -6.3333, A 0.000, B 0.000, C 0.000 }
gfCNCPoint5[6389] = {X 249.1857, Y 22.7034, Z -6.3333, A 0.000, B 0.000, C 0.000 }
gfCNCPoint5[6390] = {X 250.4352, Y 22.7777, Z -6.3333, A 0.000, B 0.000, C 0.000 }
gfCNCPoint5[6391] = {X 251.6867, Y 22.7960, Z -6.3333, A 0.000, B 0.000, C 0.000 }
gfCNCPoint5[6392] = {X 252.9776, Y 22.7960, Z -6.3333, A 0.000, B 0.000, C 0.000 }
gfCNCPoint5[6393] = {X 256.9624, Y 22.4474, Z -6.3333, A 0.000, B 0.000, C 0.000 }
gfCNCPoint5[6394] = {X 248.9928, Y 22.5274, Z -6.3333, A 0.000, B 0.000, C 0.000 }
gfCNCPoint5[6395] = {X 252.9776, Y 22.8760, Z -6.3333, A 0.000, B 0.000, C 0.000 }
gfCNCPoint5[6396] = {X 257.7315, Y 22.8760, Z -6.3333, A 0.000, B 0.000, C 0.000 }
gfCNCPoint5[6397] = {X 257.7315, Y 19.4617, Z -6.3333, A 0.000, B 0.000, C 0.000 }
gfCNCPoint5[6398] = {X 251.5267, Y 19.4617, Z -6.3333, A 0.000, B 0.000, C 0.000 }
gfCNCPoint5[6399] = {X 250.8343, Y 19.4726, Z -6.3333, A 0.000, B 0.000, C 0.000 }
gfCNCPoint5[6400] = {X 249.7949, Y 19.5478, Z -6.3333, A 0.000, B 0.000, C 0.000 }
gfCNCPoint5[6401] = {X 248.7763, Y 19.7682, Z -6.3333, A 0.000, B 0.000, C 0.000 }
gfCNCPoint5[6402] = {X 248.4828, Y 19.9234, Z -6.3333, A 0.000, B 0.000, C 0.000 }
gfCNCPoint5[6403] = {X 248.3081, Y 20.2058, Z -6.3333, A 0.000, B 0.000, C 0.000 }
gfCNCPoint5[6404] = {X 248.1533, Y 20.9889, Z -6.3333, A 0.000, B 0.000, C 0.000 }
gfCNCPoint5[6405] = {X 248.1465, Y 21.7871, Z -6.3333, A 0.000, B 0.000, C 0.000 }
gfCNCPoint5[6406] = {X 248.2880, Y 22.5727, Z -6.3333, A 0.000, B 0.000, C 0.000 }
gfCNCPoint5[6407] = {X 248.3067, Y 22.5961, Z -6.3333, A 0.000, B 0.000, C 0.000 }
gfCNCPoint5[6408] = {X 248.3330, Y 22.6053, Z -6.3333, A 0.000, B 0.000, C 0.000 }
gfCNCPoint5[6409] = {X 248.7505, Y 22.7208, Z -6.3333, A 0.000, B 0.000, C 0.000 }
gfCNCPoint5[6410] = {X 249.1792, Y 22.7831, Z -6.3333, A 0.000, B 0.000, C 0.000 }
gfCNCPoint5[6411] = {X 250.4321, Y 22.8576, Z -6.3333, A 0.000, B 0.000, C 0.000 }
gfCNCPoint5[6412] = {X 251.6870, Y 22.8760, Z -6.3333, A 0.000, B 0.000, C 0.000 }
gfCNCPoint5[6413] = {X 252.9776, Y 22.8760, Z -6.3333, A 0.000, B 0.000, C 0.000 }
gfCNCPoint5[6414] = {X 256.9624, Y 22.5274, Z -6.3333, A 0.000, B 0.000, C 0.000 }
gfCNCPoint5[6415] = {X 248.9928, Y 22.6074, Z -6.3333, A 0.000, B 0.000, C 0.000 }
gfCNCPoint5[6416] = {X 252.9776, Y 22.9560, Z -6.3333, A 0.000, B 0.000, C 0.000 }
gfCNCPoint5[6417] = {X 257.8115, Y 22.9560, Z -6.3333, A 0.000, B 0.000, C 0.000 }
gfCNCPoint5[6418] = {X 257.8111, Y 19.3817, Z -6.3333, A 0.000, B 0.000, C 0.000 }
gfCNCPoint5[6419] = {X 251.5261, Y 19.3817, Z -6.3333, A 0.000, B 0.000, C 0.000 }
gfCNCPoint5[6420] = {X 250.8336, Y 19.3926, Z -6.3333, A 0.000, B 0.000, C 0.000 }
gfCNCPoint5[6421] = {X 249.7844, Y 19.4685, Z -6.3333, A 0.000, B 0.000, C 0.000 }
gfCNCPoint5[6422] = {X 248.7562, Y 19.6907, Z -6.3333, A 0.000, B 0.000, C 0.000 }
gfCNCPoint5[6423] = {X 248.4272, Y 19.8659, Z -6.3333, A 0.000, B 0.000, C 0.000 }
gfCNCPoint5[6424] = {X 248.2314, Y 20.1831, Z -6.3333, A 0.000, B 0.000, C 0.000 }
gfCNCPoint5[6425] = {X 248.0732, Y 20.9862, Z -6.3333, A 0.000, B 0.000, C 0.000 }
gfCNCPoint5[6426] = {X 248.0678, Y 21.8048, Z -6.3333, A 0.000, B 0.000, C 0.000 }
gfCNCPoint5[6427] = {X 248.2154, Y 22.6099, Z -6.3333, A 0.000, B 0.000, C 0.000 }
gfCNCPoint5[6428] = {X 248.2584, Y 22.6638, Z -6.3333, A 0.000, B 0.000, C 0.000 }
gfCNCPoint5[6429] = {X 248.7089, Y 22.7937, Z -6.3333, A 0.000, B 0.000, C 0.000 }
gfCNCPoint5[6430] = {X 249.1727, Y 22.8628, Z -6.3333, A 0.000, B 0.000, C 0.000 }
gfCNCPoint5[6431] = {X 250.4290, Y 22.9375, Z -6.3333, A 0.000, B 0.000, C 0.000 }
gfCNCPoint5[6432] = {X 251.6873, Y 22.9560, Z -6.3333, A 0.000, B 0.000, C 0.000 }
gfCNCPoint5[6433] = {X 252.9776, Y 22.9560, Z -6.3333, A 0.000, B 0.000, C 0.000 }
gfCNCPoint5[6434] = {X 256.9624, Y 22.6074, Z -6.3333, A 0.000, B 0.000, C 0.000 }
gfCNCPoint5[6435] = {X 256.9624, Y 22.6074, Z -3.3333, A 0.000, B 0.000, C 0.000 }
gfCNCPoint5[6436] = {X 256.9624, Y 22.6074, Z 11.0000, A 0.000, B 0.000, C 0.000 }
gfCNCPoint5[6437] = {X 188.4986, Y 19.4681, Z 11.0000, A 0.000, B 0.000, C 0.000 }
gfCNCPoint5[6438] = {X 188.4986, Y 19.4681, Z -2.5000, A 0.000, B 0.000, C 0.000 }
gfCNCPoint5[6439] = {X 188.3884, Y 19.4291, Z -2.5313, A 0.000, B 0.000, C 0.000 }
gfCNCPoint5[6440] = {X 187.7714, Y 19.3606, Z -2.6977, A 0.000, B 0.000, C 0.000 }
gfCNCPoint5[6441] = {X 186.9109, Y 19.2606, Z -2.9298, A 0.000, B 0.000, C 0.000 }
gfCNCPoint5[6442] = {X 184.5930, Y 19.3681, Z -3.5515, A 0.000, B 0.000, C 0.000 }
gfCNCPoint5[6443] = {X 183.7426, Y 19.5479, Z -3.7844, A 0.000, B 0.000, C 0.000 }
gfCNCPoint5[6444] = {X 183.0434, Y 19.6904, Z -3.9756, A 0.000, B 0.000, C 0.000 }
gfCNCPoint5[6445] = {X 182.0226, Y 20.0619, Z -4.2667, A 0.000, B 0.000, C 0.000 }
gfCNCPoint5[6446] = {X 181.3954, Y 20.4021, Z -4.4579, A 0.000, B 0.000, C 0.000 }
gfCNCPoint5[6447] = {X 181.3394, Y 20.9137, Z -4.5958, A 0.000, B 0.000, C 0.000 }
gfCNCPoint5[6448] = {X 180.8652, Y 22.1256, Z -4.9445, A 0.000, B 0.000, C 0.000 }
gfCNCPoint5[6449] = {X 180.5592, Y 22.5394, Z -5.0824, A 0.000, B 0.000, C 0.000 }
gfCNCPoint5[6450] = {X 182.2919, Y 22.3335, Z -5.5500, A 0.000, B 0.000, C 0.000 }
gfCNCPoint5[6451] = {X 182.5945, Y 22.3089, Z -5.6313, A 0.000, B 0.000, C 0.000 }
gfCNCPoint5[6452] = {X 184.3413, Y 22.2328, Z -6.0998, A 0.000, B 0.000, C 0.000 }
gfCNCPoint5[6453] = {X 184.7768, Y 22.2177, Z -6.2166, A 0.000, B 0.000, C 0.000 }
gfCNCPoint5[6454] = {X 185.2121, Y 22.1993, Z -6.3333, A 0.000, B 0.000, C 0.000 }
gfCNCPoint5[6455] = {X 187.5423, Y 22.0769, Z -6.3333, A 0.000, B 0.000, C 0.000 }
gfCNCPoint5[6456] = {X 189.8695, Y 21.9070, Z -6.3333, A 0.000, B 0.000, C 0.000 }
gfCNCPoint5[6457] = {X 190.4710, Y 21.8304, Z -6.3333, A 0.000, B 0.000, C 0.000 }
gfCNCPoint5[6458] = {X 191.0581, Y 21.6792, Z -6.3333, A 0.000, B 0.000, C 0.000 }
gfCNCPoint5[6459] = {X 191.0678, Y 21.1638, Z -6.3333, A 0.000, B 0.000, C 0.000 }
gfCNCPoint5[6460] = {X 190.8721, Y 20.6868, Z -6.3333, A 0.000, B 0.000, C 0.000 }
gfCNCPoint5[6461] = {X 190.5033, Y 20.3267, Z -6.3333, A 0.000, B 0.000, C 0.000 }
gfCNCPoint5[6462] = {X 189.6458, Y 19.8660, Z -6.3333, A 0.000, B 0.000, C 0.000 }
gfCNCPoint5[6463] = {X 188.7280, Y 19.5414, Z -6.3333, A 0.000, B 0.000, C 0.000 }
gfCNCPoint5[6464] = {X 187.7714, Y 19.3606, Z -6.3333, A 0.000, B 0.000, C 0.000 }
gfCNCPoint5[6465] = {X 186.4243, Y 19.2775, Z -6.3333, A 0.000, B 0.000, C 0.000 }
gfCNCPoint5[6466] = {X 185.0761, Y 19.3401, Z -6.3333, A 0.000, B 0.000, C 0.000 }
gfCNCPoint5[6467] = {X 183.7426, Y 19.5479, Z -6.3333, A 0.000, B 0.000, C 0.000 }
gfCNCPoint5[6468] = {X 182.5373, Y 19.8880, Z -6.3333, A 0.000, B 0.000, C 0.000 }
gfCNCPoint5[6469] = {X 181.3954, Y 20.4021, Z -6.3333, A 0.000, B 0.000, C 0.000 }
gfCNCPoint5[6470] = {X 181.2441, Y 21.1601, Z -6.3333, A 0.000, B 0.000, C 0.000 }
gfCNCPoint5[6471] = {X 180.9624, Y 21.8800, Z -6.3333, A 0.000, B 0.000, C 0.000 }
gfCNCPoint5[6472] = {X 180.5592, Y 22.5394, Z -6.3333, A 0.000, B 0.000, C 0.000 }
gfCNCPoint5[6473] = {X 182.4474, Y 22.3508, Z -6.3333, A 0.000, B 0.000, C 0.000 }
gfCNCPoint5[6474] = {X 184.3413, Y 22.2328, Z -6.3333, A 0.000, B 0.000, C 0.000 }
gfCNCPoint5[6475] = {X 184.7767, Y 22.2169, Z -6.3333, A 0.000, B 0.000, C 0.000 }
gfCNCPoint5[6476] = {X 185.2121, Y 22.1993, Z -6.3333, A 0.000, B 0.000, C 0.000 }
gfCNCPoint5[6477] = {X 181.2196, Y 22.0994, Z -6.3333, A 0.000, B 0.000, C 0.000 }
gfCNCPoint5[6478] = {X 185.2155, Y 22.2792, Z -6.3333, A 0.000, B 0.000, C 0.000 }
gfCNCPoint5[6479] = {X 187.5451, Y 22.1568, Z -6.3333, A 0.000, B 0.000, C 0.000 }
gfCNCPoint5[6480] = {X 189.8716, Y 21.9870, Z -6.3333, A 0.000, B 0.000, C 0.000 }
gfCNCPoint5[6481] = {X 190.5065, Y 21.9050, Z -6.3333, A 0.000, B 0.000, C 0.000 }
gfCNCPoint5[6482] = {X 191.1253, Y 21.7412, Z -6.3333, A 0.000, B 0.000, C 0.000 }
gfCNCPoint5[6483] = {X 191.1517, Y 21.1790, Z -6.3333, A 0.000, B 0.000, C 0.000 }
gfCNCPoint5[6484] = {X 190.9469, Y 20.6548, Z -6.3333, A 0.000, B 0.000, C 0.000 }
gfCNCPoint5[6485] = {X 190.5465, Y 20.2593, Z -6.3333, A 0.000, B 0.000, C 0.000 }
gfCNCPoint5[6486] = {X 189.6787, Y 19.7931, Z -6.3333, A 0.000, B 0.000, C 0.000 }
gfCNCPoint5[6487] = {X 188.7501, Y 19.4645, Z -6.3333, A 0.000, B 0.000, C 0.000 }
gfCNCPoint5[6488] = {X 187.7823, Y 19.2813, Z -6.3333, A 0.000, B 0.000, C 0.000 }
gfCNCPoint5[6489] = {X 186.4270, Y 19.1975, Z -6.3333, A 0.000, B 0.000, C 0.000 }
gfCNCPoint5[6490] = {X 185.0706, Y 19.2603, Z -6.3333, A 0.000, B 0.000, C 0.000 }
gfCNCPoint5[6491] = {X 183.7289, Y 19.4690, Z -6.3333, A 0.000, B 0.000, C 0.000 }
gfCNCPoint5[6492] = {X 182.4919, Y 19.8194, Z -6.3333, A 0.000, B 0.000, C 0.000 }
gfCNCPoint5[6493] = {X 181.3215, Y 20.3512, Z -6.3333, A 0.000, B 0.000, C 0.000 }
gfCNCPoint5[6494] = {X 181.1592, Y 21.1708, Z -6.3333, A 0.000, B 0.000, C 0.000 }
gfCNCPoint5[6495] = {X 180.8422, Y 21.9439, Z -6.3333, A 0.000, B 0.000, C 0.000 }
gfCNCPoint5[6496] = {X 180.3822, Y 22.6414, Z -6.3333, A 0.000, B 0.000, C 0.000 }
gfCNCPoint5[6497] = {X 182.3592, Y 22.4382, Z -6.3333, A 0.000, B 0.000, C 0.000 }
gfCNCPoint5[6498] = {X 184.3427, Y 22.3128, Z -6.3333, A 0.000, B 0.000, C 0.000 }
gfCNCPoint5[6499] = {X 184.7791, Y 22.2968, Z -6.3333, A 0.000, B 0.000, C 0.000 }
gfCNCPoint5[6500] = {X 185.2155, Y 22.2792, Z -6.3333, A 0.000, B 0.000, C 0.000 }
gfCNCPoint5[6501] = {X 189.1820, Y 21.7624, Z -6.3333, A 0.000, B 0.000, C 0.000 }
gfCNCPoint5[6502] = {X 181.2229, Y 22.1793, Z -6.3333, A 0.000, B 0.000, C 0.000 }
gfCNCPoint5[6503] = {X 185.2189, Y 22.3591, Z -6.3333, A 0.000, B 0.000, C 0.000 }
gfCNCPoint5[6504] = {X 187.5497, Y 22.2367, Z -6.3333, A 0.000, B 0.000, C 0.000 }
gfCNCPoint5[6505] = {X 189.8775, Y 22.0668, Z -6.3333, A 0.000, B 0.000, C 0.000 }
gfCNCPoint5[6506] = {X 190.5431, Y 21.9793, Z -6.3333, A 0.000, B 0.000, C 0.000 }
gfCNCPoint5[6507] = {X 191.1910, Y 21.8033, Z -6.3333, A 0.000, B 0.000, C 0.000 }
gfCNCPoint5[6508] = {X 191.2486, Y 21.3477, Z -6.3333, A 0.000, B 0.000, C 0.000 }
gfCNCPoint5[6509] = {X 191.1591, Y 20.8973, Z -6.3333, A 0.000, B 0.000, C 0.000 }
gfCNCPoint5[6510] = {X 190.9316, Y 20.4984, Z -6.3333, A 0.000, B 0.000, C 0.000 }
gfCNCPoint5[6511] = {X 190.5896, Y 20.1919, Z -6.3333, A 0.000, B 0.000, C 0.000 }
gfCNCPoint5[6512] = {X 189.7111, Y 19.7199, Z -6.3333, A 0.000, B 0.000, C 0.000 }
gfCNCPoint5[6513] = {X 188.7710, Y 19.3873, Z -6.3333, A 0.000, B 0.000, C 0.000 }
gfCNCPoint5[6514] = {X 187.7911, Y 19.2018, Z -6.3333, A 0.000, B 0.000, C 0.000 }
gfCNCPoint5[6515] = {X 186.4273, Y 19.1175, Z -6.3333, A 0.000, B 0.000, C 0.000 }
gfCNCPoint5[6516] = {X 185.0625, Y 19.1807, Z -6.3333, A 0.000, B 0.000, C 0.000 }
gfCNCPoint5[6517] = {X 183.7123, Y 19.3907, Z -6.3333, A 0.000, B 0.000, C 0.000 }
gfCNCPoint5[6518] = {X 182.4465, Y 19.7509, Z -6.3333, A 0.000, B 0.000, C 0.000 }
gfCNCPoint5[6519] = {X 181.2500, Y 20.2993, Z -6.3333, A 0.000, B 0.000, C 0.000 }
gfCNCPoint5[6520] = {X 181.2397, Y 20.3530, Z -6.3333, A 0.000, B 0.000, C 0.000 }
gfCNCPoint5[6521] = {X 181.0598, Y 21.2186, Z -6.3333, A 0.000, B 0.000, C 0.000 }
gfCNCPoint5[6522] = {X 180.7042, Y 22.0280, Z -6.3333, A 0.000, B 0.000, C 0.000 }
gfCNCPoint5[6523] = {X 180.1886, Y 22.7462, Z -6.3333, A 0.000, B 0.000, C 0.000 }
gfCNCPoint5[6524] = {X 182.2635, Y 22.5266, Z -6.3333, A 0.000, B 0.000, C 0.000 }
gfCNCPoint5[6525] = {X 184.3458, Y 22.3928, Z -6.3333, A 0.000, B 0.000, C 0.000 }
gfCNCPoint5[6526] = {X 184.7824, Y 22.3768, Z -6.3333, A 0.000, B 0.000, C 0.000 }
gfCNCPoint5[6527] = {X 185.2189, Y 22.3591, Z -6.3333, A 0.000, B 0.000, C 0.000 }
gfCNCPoint5[6528] = {X 189.1854, Y 21.8423, Z -6.3333, A 0.000, B 0.000, C 0.000 }
gfCNCPoint5[6529] = {X 181.2263, Y 22.2593, Z -6.3333, A 0.000, B 0.000, C 0.000 }
gfCNCPoint5[6530] = {X 185.2223, Y 22.4391, Z -6.3333, A 0.000, B 0.000, C 0.000 }
gfCNCPoint5[6531] = {X 187.5543, Y 22.3165, Z -6.3333, A 0.000, B 0.000, C 0.000 }
gfCNCPoint5[6532] = {X 189.8833, Y 22.1466, Z -6.3333, A 0.000, B 0.000, C 0.000 }
gfCNCPoint5[6533] = {X 190.5791, Y 22.0536, Z -6.3333, A 0.000, B 0.000, C 0.000 }
gfCNCPoint5[6534] = {X 191.2555, Y 21.8655, Z -6.3333, A 0.000, B 0.000, C 0.000 }
gfCNCPoint5[6535] = {X 191.3294, Y 21.3760, Z -6.3333, A 0.000, B 0.000, C 0.000 }
gfCNCPoint5[6536] = {X 191.2412, Y 20.8888, Z -6.3333, A 0.000, B 0.000, C 0.000 }
gfCNCPoint5[6537] = {X 191.0004, Y 20.4562, Z -6.3333, A 0.000, B 0.000, C 0.000 }
gfCNCPoint5[6538] = {X 190.6327, Y 20.1246, Z -6.3333, A 0.000, B 0.000, C 0.000 }
gfCNCPoint5[6539] = {X 189.7435, Y 19.6468, Z -6.3333, A 0.000, B 0.000, C 0.000 }
gfCNCPoint5[6540] = {X 188.7918, Y 19.3101, Z -6.3333, A 0.000, B 0.000, C 0.000 }
gfCNCPoint5[6541] = {X 187.7999, Y 19.1223, Z -6.3333, A 0.000, B 0.000, C 0.000 }
gfCNCPoint5[6542] = {X 186.4277, Y 19.0375, Z -6.3333, A 0.000, B 0.000, C 0.000 }
gfCNCPoint5[6543] = {X 185.0543, Y 19.1011, Z -6.3333, A 0.000, B 0.000, C 0.000 }
gfCNCPoint5[6544] = {X 183.6958, Y 19.3125, Z -6.3333, A 0.000, B 0.000, C 0.000 }
gfCNCPoint5[6545] = {X 182.4009, Y 19.6824, Z -6.3333, A 0.000, B 0.000, C 0.000 }
gfCNCPoint5[6546] = {X 181.1785, Y 20.2476, Z -6.3333, A 0.000, B 0.000, C 0.000 }
gfCNCPoint5[6547] = {X 181.1605, Y 20.3414, Z -6.3333, A 0.000, B 0.000, C 0.000 }
gfCNCPoint5[6548] = {X 180.9651, Y 21.2476, Z -6.3333, A 0.000, B 0.000, C 0.000 }
gfCNCPoint5[6549] = {X 180.5738, Y 22.0880, Z -6.3333, A 0.000, B 0.000, C 0.000 }
gfCNCPoint5[6550] = {X 180.0062, Y 22.8209, Z -6.3333, A 0.000, B 0.000, C 0.000 }
gfCNCPoint5[6551] = {X 180.1925, Y 22.8263, Z -6.3333, A 0.000, B 0.000, C 0.000 }
gfCNCPoint5[6552] = {X 182.2670, Y 22.6066, Z -6.3333, A 0.000, B 0.000, C 0.000 }
gfCNCPoint5[6553] = {X 184.3489, Y 22.4727, Z -6.3333, A 0.000, B 0.000, C 0.000 }
gfCNCPoint5[6554] = {X 184.7856, Y 22.4567, Z -6.3333, A 0.000, B 0.000, C 0.000 }
gfCNCPoint5[6555] = {X 185.2223, Y 22.4391, Z -6.3333, A 0.000, B 0.000, C 0.000 }
gfCNCPoint5[6556] = {X 189.1887, Y 21.9222, Z -6.3333, A 0.000, B 0.000, C 0.000 }
gfCNCPoint5[6557] = {X 181.2297, Y 22.3392, Z -6.3333, A 0.000, B 0.000, C 0.000 }
gfCNCPoint5[6558] = {X 185.2257, Y 22.5190, Z -6.3333, A 0.000, B 0.000, C 0.000 }
gfCNCPoint5[6559] = {X 187.5589, Y 22.3964, Z -6.3333, A 0.000, B 0.000, C 0.000 }
gfCNCPoint5[6560] = {X 189.8892, Y 22.2264, Z -6.3333, A 0.000, B 0.000, C 0.000 }
gfCNCPoint5[6561] = {X 190.6146, Y 22.1280, Z -6.3333, A 0.000, B 0.000, C 0.000 }
gfCNCPoint5[6562] = {X 191.3188, Y 21.9278, Z -6.3333, A 0.000, B 0.000, C 0.000 }
gfCNCPoint5[6563] = {X 191.4095, Y 21.4045, Z -6.3333, A 0.000, B 0.000, C 0.000 }
gfCNCPoint5[6564] = {X 191.3231, Y 20.8805, Z -6.3333, A 0.000, B 0.000, C 0.000 }
gfCNCPoint5[6565] = {X 191.0691, Y 20.4141, Z -6.3333, A 0.000, B 0.000, C 0.000 }
gfCNCPoint5[6566] = {X 190.6759, Y 20.0572, Z -6.3333, A 0.000, B 0.000, C 0.000 }
gfCNCPoint5[6567] = {X 189.7758, Y 19.5736, Z -6.3333, A 0.000, B 0.000, C 0.000 }
gfCNCPoint5[6568] = {X 188.8126, Y 19.2328, Z -6.3333, A 0.000, B 0.000, C 0.000 }
gfCNCPoint5[6569] = {X 187.8088, Y 19.0428, Z -6.3333, A 0.000, B 0.000, C 0.000 }
gfCNCPoint5[6570] = {X 186.4280, Y 18.9575, Z -6.3333, A 0.000, B 0.000, C 0.000 }
gfCNCPoint5[6571] = {X 185.0462, Y 19.0215, Z -6.3333, A 0.000, B 0.000, C 0.000 }
gfCNCPoint5[6572] = {X 183.6792, Y 19.2342, Z -6.3333, A 0.000, B 0.000, C 0.000 }
gfCNCPoint5[6573] = {X 182.3553, Y 19.6141, Z -6.3333, A 0.000, B 0.000, C 0.000 }
gfCNCPoint5[6574] = {X 181.1070, Y 20.1960, Z -6.3333, A 0.000, B 0.000, C 0.000 }
gfCNCPoint5[6575] = {X 181.0812, Y 20.3298, Z -6.3333, A 0.000, B 0.000, C 0.000 }
gfCNCPoint5[6576] = {X 180.8699, Y 21.2784, Z -6.3333, A 0.000, B 0.000, C 0.000 }
gfCNCPoint5[6577] = {X 180.4402, Y 22.1501, Z -6.3333, A 0.000, B 0.000, C 0.000 }
gfCNCPoint5[6578] = {X 179.8165, Y 22.8954, Z -6.3333, A 0.000, B 0.000, C 0.000 }
gfCNCPoint5[6579] = {X 180.1964, Y 22.9065, Z -6.3333, A 0.000, B 0.000, C 0.000 }
gfCNCPoint5[6580] = {X 182.2705, Y 22.6865, Z -6.3333, A 0.000, B 0.000, C 0.000 }
gfCNCPoint5[6581] = {X 184.3520, Y 22.5526, Z -6.3333, A 0.000, B 0.000, C 0.000 }
gfCNCPoint5[6582] = {X 184.7889, Y 22.5366, Z -6.3333, A 0.000, B 0.000, C 0.000 }
gfCNCPoint5[6583] = {X 185.2257, Y 22.5190, Z -6.3333, A 0.000, B 0.000, C 0.000 }
gfCNCPoint5[6584] = {X 189.1921, Y 22.0021, Z -6.3333, A 0.000, B 0.000, C 0.000 }
gfCNCPoint5[6585] = {X 185.1540, Y 22.6021, Z -6.3333, A 0.000, B 0.000, C 0.000 }
gfCNCPoint5[6586] = {X 185.2290, Y 22.5989, Z -6.3333, A 0.000, B 0.000, C 0.000 }
gfCNCPoint5[6587] = {X 187.5635, Y 22.4763, Z -6.3333, A 0.000, B 0.000, C 0.000 }
gfCNCPoint5[6588] = {X 189.8950, Y 22.3061, Z -6.3333, A 0.000, B 0.000, C 0.000 }
gfCNCPoint5[6589] = {X 190.6497, Y 22.2024, Z -6.3333, A 0.000, B 0.000, C 0.000 }
gfCNCPoint5[6590] = {X 191.3812, Y 21.9901, Z -6.3333, A 0.000, B 0.000, C 0.000 }
gfCNCPoint5[6591] = {X 191.4892, Y 21.4334, Z -6.3333, A 0.000, B 0.000, C 0.000 }
gfCNCPoint5[6592] = {X 191.4048, Y 20.8726, Z -6.3333, A 0.000, B 0.000, C 0.000 }
gfCNCPoint5[6593] = {X 191.1379, Y 20.3722, Z -6.3333, A 0.000, B 0.000, C 0.000 }
gfCNCPoint5[6594] = {X 190.7190, Y 19.9898, Z -6.3333, A 0.000, B 0.000, C 0.000 }
gfCNCPoint5[6595] = {X 189.8082, Y 19.5005, Z -6.3333, A 0.000, B 0.000, C 0.000 }
gfCNCPoint5[6596] = {X 188.8335, Y 19.1556, Z -6.3333, A 0.000, B 0.000, C 0.000 }
gfCNCPoint5[6597] = {X 187.8176, Y 18.9632, Z -6.3333, A 0.000, B 0.000, C 0.000 }
gfCNCPoint5[6598] = {X 186.4284, Y 18.8775, Z -6.3333, A 0.000, B 0.000, C 0.000 }
gfCNCPoint5[6599] = {X 185.0380, Y 18.9420, Z -6.3333, A 0.000, B 0.000, C 0.000 }
gfCNCPoint5[6600] = {X 183.6627, Y 19.1559, Z -6.3333, A 0.000, B 0.000, C 0.000 }
gfCNCPoint5[6601] = {X 182.3097, Y 19.5457, Z -6.3333, A 0.000, B 0.000, C 0.000 }
gfCNCPoint5[6602] = {X 181.0354, Y 20.1447, Z -6.3333, A 0.000, B 0.000, C 0.000 }
gfCNCPoint5[6603] = {X 181.0020, Y 20.3183, Z -6.3333, A 0.000, B 0.000, C 0.000 }
gfCNCPoint5[6604] = {X 180.8538, Y 21.0695, Z -6.3333, A 0.000, B 0.000, C 0.000 }
gfCNCPoint5[6605] = {X 180.5651, Y 21.7787, Z -6.3333, A 0.000, B 0.000, C 0.000 }
gfCNCPoint5[6606] = {X 180.1466, Y 22.4199, Z -6.3333, A 0.000, B 0.000, C 0.000 }
gfCNCPoint5[6607] = {X 179.6136, Y 22.9696, Z -6.3333, A 0.000, B 0.000, C 0.000 }
gfCNCPoint5[6608] = {X 180.2003, Y 22.9866, Z -6.3333, A 0.000, B 0.000, C 0.000 }
gfCNCPoint5[6609] = {X 182.2741, Y 22.7665, Z -6.3333, A 0.000, B 0.000, C 0.000 }
gfCNCPoint5[6610] = {X 184.3552, Y 22.6326, Z -6.3333, A 0.000, B 0.000, C 0.000 }
gfCNCPoint5[6611] = {X 184.7921, Y 22.6166, Z -6.3333, A 0.000, B 0.000, C 0.000 }
gfCNCPoint5[6612] = {X 185.2290, Y 22.5989, Z -6.3333, A 0.000, B 0.000, C 0.000 }
gfCNCPoint5[6613] = {X 185.1445, Y 20.6007, Z -6.3333, A 0.000, B 0.000, C 0.000 }
gfCNCPoint5[6614] = {X 185.1445, Y 20.6007, Z -3.3333, A 0.000, B 0.000, C 0.000 }
gfCNCPoint5[6615] = {X 185.1445, Y 20.6007, Z 11.0000, A 0.000, B 0.000, C 0.000 }
gfCNCPoint5[6616] = {X 186.2272, Y 37.9118, Z 11.0000, A 0.000, B 0.000, C 0.000 }
gfCNCPoint5[6617] = {X 186.2272, Y 37.9118, Z -2.5000, A 0.000, B 0.000, C 0.000 }
gfCNCPoint5[6618] = {X 187.5901, Y 37.8319, Z -2.8658, A 0.000, B 0.000, C 0.000 }
gfCNCPoint5[6619] = {X 189.4174, Y 37.3853, Z -3.3699, A 0.000, B 0.000, C 0.000 }
gfCNCPoint5[6620] = {X 190.9814, Y 36.7125, Z -3.8261, A 0.000, B 0.000, C 0.000 }
gfCNCPoint5[6621] = {X 191.6907, Y 36.3242, Z -4.0427, A 0.000, B 0.000, C 0.000 }
gfCNCPoint5[6622] = {X 192.4467, Y 35.8117, Z -4.2874, A 0.000, B 0.000, C 0.000 }
gfCNCPoint5[6623] = {X 192.4700, Y 35.2976, Z -4.4253, A 0.000, B 0.000, C 0.000 }
gfCNCPoint5[6624] = {X 192.6311, Y 34.6355, Z -4.6079, A 0.000, B 0.000, C 0.000 }
gfCNCPoint5[6625] = {X 192.8467, Y 34.1681, Z -4.7458, A 0.000, B 0.000, C 0.000 }
gfCNCPoint5[6626] = {X 192.7389, Y 34.1932, Z -4.7755, A 0.000, B 0.000, C 0.000 }
gfCNCPoint5[6627] = {X 191.4073, Y 34.4435, Z -5.1386, A 0.000, B 0.000, C 0.000 }
gfCNCPoint5[6628] = {X 190.5822, Y 34.5497, Z -5.3615, A 0.000, B 0.000, C 0.000 }
gfCNCPoint5[6629] = {X 189.2271, Y 34.6449, Z -5.7255, A 0.000, B 0.000, C 0.000 }
gfCNCPoint5[6630] = {X 186.9627, Y 34.7839, Z -6.3333, A 0.000, B 0.000, C 0.000 }
gfCNCPoint5[6631] = {X 182.5706, Y 35.0536, Z -6.3333, A 0.000, B 0.000, C 0.000 }
gfCNCPoint5[6632] = {X 181.8152, Y 35.1408, Z -6.3333, A 0.000, B 0.000, C 0.000 }
gfCNCPoint5[6633] = {X 181.0734, Y 35.3082, Z -6.3333, A 0.000, B 0.000, C 0.000 }
gfCNCPoint5[6634] = {X 181.0653, Y 35.3824, Z -6.3333, A 0.000, B 0.000, C 0.000 }
gfCNCPoint5[6635] = {X 181.0654, Y 35.4570, Z -6.3333, A 0.000, B 0.000, C 0.000 }
gfCNCPoint5[6636] = {X 181.1580, Y 35.9997, Z -6.3333, A 0.000, B 0.000, C 0.000 }
gfCNCPoint5[6637] = {X 181.4150, Y 36.4867, Z -6.3333, A 0.000, B 0.000, C 0.000 }
gfCNCPoint5[6638] = {X 181.8108, Y 36.8694, Z -6.3333, A 0.000, B 0.000, C 0.000 }
gfCNCPoint5[6639] = {X 182.4283, Y 37.2223, Z -6.3333, A 0.000, B 0.000, C 0.000 }
gfCNCPoint5[6640] = {X 183.0886, Y 37.4869, Z -6.3333, A 0.000, B 0.000, C 0.000 }
gfCNCPoint5[6641] = {X 184.4949, Y 37.8008, Z -6.3333, A 0.000, B 0.000, C 0.000 }
gfCNCPoint5[6642] = {X 185.9312, Y 37.9167, Z -6.3333, A 0.000, B 0.000, C 0.000 }
gfCNCPoint5[6643] = {X 187.3696, Y 37.8324, Z -6.3333, A 0.000, B 0.000, C 0.000 }
gfCNCPoint5[6644] = {X 188.7825, Y 37.5495, Z -6.3333, A 0.000, B 0.000, C 0.000 }
gfCNCPoint5[6645] = {X 190.1425, Y 37.0734, Z -6.3333, A 0.000, B 0.000, C 0.000 }
gfCNCPoint5[6646] = {X 191.3245, Y 36.4972, Z -6.3333, A 0.000, B 0.000, C 0.000 }
gfCNCPoint5[6647] = {X 192.4467, Y 35.8117, Z -6.3333, A 0.000, B 0.000, C 0.000 }
gfCNCPoint5[6648] = {X 192.5669, Y 34.9705, Z -6.3333, A 0.000, B 0.000, C 0.000 }
gfCNCPoint5[6649] = {X 192.8467, Y 34.1681, Z -6.3333, A 0.000, B 0.000, C 0.000 }
gfCNCPoint5[6650] = {X 192.7389, Y 34.1932, Z -6.3333, A 0.000, B 0.000, C 0.000 }
gfCNCPoint5[6651] = {X 190.9895, Y 34.4699, Z -6.3333, A 0.000, B 0.000, C 0.000 }
gfCNCPoint5[6652] = {X 189.2271, Y 34.6449, Z -6.3333, A 0.000, B 0.000, C 0.000 }
gfCNCPoint5[6653] = {X 186.9627, Y 34.7839, Z -6.3333, A 0.000, B 0.000, C 0.000 }
gfCNCPoint5[6654] = {X 190.9565, Y 34.8078, Z -6.3333, A 0.000, B 0.000, C 0.000 }
gfCNCPoint5[6655] = {X 186.9578, Y 34.7041, Z -6.3333, A 0.000, B 0.000, C 0.000 }
gfCNCPoint5[6656] = {X 182.5657, Y 34.9737, Z -6.3333, A 0.000, B 0.000, C 0.000 }
gfCNCPoint5[6657] = {X 181.7775, Y 35.0661, Z -6.3333, A 0.000, B 0.000, C 0.000 }
gfCNCPoint5[6658] = {X 181.0044, Y 35.2448, Z -6.3333, A 0.000, B 0.000, C 0.000 }
gfCNCPoint5[6659] = {X 180.9877, Y 35.3482, Z -6.3333, A 0.000, B 0.000, C 0.000 }
gfCNCPoint5[6660] = {X 180.9854, Y 35.4530, Z -6.3333, A 0.000, B 0.000, C 0.000 }
gfCNCPoint5[6661] = {X 181.0813, Y 36.0226, Z -6.3333, A 0.000, B 0.000, C 0.000 }
gfCNCPoint5[6662] = {X 181.3504, Y 36.5339, Z -6.3333, A 0.000, B 0.000, C 0.000 }
gfCNCPoint5[6663] = {X 181.7656, Y 36.9355, Z -6.3333, A 0.000, B 0.000, C 0.000 }
gfCNCPoint5[6664] = {X 182.3935, Y 37.2944, Z -6.3333, A 0.000, B 0.000, C 0.000 }
gfCNCPoint5[6665] = {X 183.0649, Y 37.5633, Z -6.3333, A 0.000, B 0.000, C 0.000 }
gfCNCPoint5[6666] = {X 184.4822, Y 37.8798, Z -6.3333, A 0.000, B 0.000, C 0.000 }
gfCNCPoint5[6667] = {X 185.9297, Y 37.9967, Z -6.3333, A 0.000, B 0.000, C 0.000 }
gfCNCPoint5[6668] = {X 187.3795, Y 37.9118, Z -6.3333, A 0.000, B 0.000, C 0.000 }
gfCNCPoint5[6669] = {X 188.8034, Y 37.6267, Z -6.3333, A 0.000, B 0.000, C 0.000 }
gfCNCPoint5[6670] = {X 190.1741, Y 37.1469, Z -6.3333, A 0.000, B 0.000, C 0.000 }
gfCNCPoint5[6671] = {X 191.3806, Y 36.5576, Z -6.3333, A 0.000, B 0.000, C 0.000 }
gfCNCPoint5[6672] = {X 192.5249, Y 35.8552, Z -6.3333, A 0.000, B 0.000, C 0.000 }
gfCNCPoint5[6673] = {X 192.6601, Y 34.9278, Z -6.3333, A 0.000, B 0.000, C 0.000 }
gfCNCPoint5[6674] = {X 192.9922, Y 34.0514, Z -6.3333, A 0.000, B 0.000, C 0.000 }
gfCNCPoint5[6675] = {X 192.7315, Y 34.1132, Z -6.3333, A 0.000, B 0.000, C 0.000 }
gfCNCPoint5[6676] = {X 190.9841, Y 34.3899, Z -6.3333, A 0.000, B 0.000, C 0.000 }
gfCNCPoint5[6677] = {X 189.2236, Y 34.5649, Z -6.3333, A 0.000, B 0.000, C 0.000 }
gfCNCPoint5[6678] = {X 186.9578, Y 34.7041, Z -6.3333, A 0.000, B 0.000, C 0.000 }
gfCNCPoint5[6679] = {X 183.0019, Y 35.2962, Z -6.3333, A 0.000, B 0.000, C 0.000 }
gfCNCPoint5[6680] = {X 190.9516, Y 34.7280, Z -6.3333, A 0.000, B 0.000, C 0.000 }
gfCNCPoint5[6681] = {X 186.9529, Y 34.6242, Z -6.3333, A 0.000, B 0.000, C 0.000 }
gfCNCPoint5[6682] = {X 182.5608, Y 34.8939, Z -6.3333, A 0.000, B 0.000, C 0.000 }
gfCNCPoint5[6683] = {X 181.7415, Y 34.9911, Z -6.3333, A 0.000, B 0.000, C 0.000 }
gfCNCPoint5[6684] = {X 180.9386, Y 35.1807, Z -6.3333, A 0.000, B 0.000, C 0.000 }
gfCNCPoint5[6685] = {X 180.9107, Y 35.3165, Z -6.3333, A 0.000, B 0.000, C 0.000 }
gfCNCPoint5[6686] = {X 180.9054, Y 35.4551, Z -6.3333, A 0.000, B 0.000, C 0.000 }
gfCNCPoint5[6687] = {X 181.0060, Y 36.0495, Z -6.3333, A 0.000, B 0.000, C 0.000 }
gfCNCPoint5[6688] = {X 181.2870, Y 36.5827, Z -6.3333, A 0.000, B 0.000, C 0.000 }
gfCNCPoint5[6689] = {X 181.7205, Y 37.0016, Z -6.3333, A 0.000, B 0.000, C 0.000 }
gfCNCPoint5[6690] = {X 182.3588, Y 37.3664, Z -6.3333, A 0.000, B 0.000, C 0.000 }
gfCNCPoint5[6691] = {X 183.0412, Y 37.6397, Z -6.3333, A 0.000, B 0.000, C 0.000 }
gfCNCPoint5[6692] = {X 184.4696, Y 37.9588, Z -6.3333, A 0.000, B 0.000, C 0.000 }
gfCNCPoint5[6693] = {X 185.9283, Y 38.0767, Z -6.3333, A 0.000, B 0.000, C 0.000 }
gfCNCPoint5[6694] = {X 187.3893, Y 37.9912, Z -6.3333, A 0.000, B 0.000, C 0.000 }
gfCNCPoint5[6695] = {X 188.8244, Y 37.7039, Z -6.3333, A 0.000, B 0.000, C 0.000 }
gfCNCPoint5[6696] = {X 190.2057, Y 37.2204, Z -6.3333, A 0.000, B 0.000, C 0.000 }
gfCNCPoint5[6697] = {X 191.4370, Y 36.6179, Z -6.3333, A 0.000, B 0.000, C 0.000 }
gfCNCPoint5[6698] = {X 192.6036, Y 35.8983, Z -6.3333, A 0.000, B 0.000, C 0.000 }
gfCNCPoint5[6699] = {X 192.6772, Y 35.2165, Z -6.3333, A 0.000, B 0.000, C 0.000 }
gfCNCPoint5[6700] = {X 192.8598, Y 34.5555, Z -6.3333, A 0.000, B 0.000, C 0.000 }
gfCNCPoint5[6701] = {X 193.1465, Y 33.9326, Z -6.3333, A 0.000, B 0.000, C 0.000 }
gfCNCPoint5[6702] = {X 192.7149, Y 34.0349, Z -6.3333, A 0.000, B 0.000, C 0.000 }
gfCNCPoint5[6703] = {X 190.9731, Y 34.3107, Z -6.3333, A 0.000, B 0.000, C 0.000 }
gfCNCPoint5[6704] = {X 189.2183, Y 34.4851, Z -6.3333, A 0.000, B 0.000, C 0.000 }
gfCNCPoint5[6705] = {X 186.9529, Y 34.6242, Z -6.3333, A 0.000, B 0.000, C 0.000 }
gfCNCPoint5[6706] = {X 182.9970, Y 35.2164, Z -6.3333, A 0.000, B 0.000, C 0.000 }
gfCNCPoint5[6707] = {X 190.9467, Y 34.6481, Z -6.3333, A 0.000, B 0.000, C 0.000 }
gfCNCPoint5[6708] = {X 186.9480, Y 34.5444, Z -6.3333, A 0.000, B 0.000, C 0.000 }
gfCNCPoint5[6709] = {X 182.5558, Y 34.8140, Z -6.3333, A 0.000, B 0.000, C 0.000 }
gfCNCPoint5[6710] = {X 181.7067, Y 34.9161, Z -6.3333, A 0.000, B 0.000, C 0.000 }
gfCNCPoint5[6711] = {X 180.8753, Y 35.1162, Z -6.3333, A 0.000, B 0.000, C 0.000 }
gfCNCPoint5[6712] = {X 180.8342, Y 35.2844, Z -6.3333, A 0.000, B 0.000, C 0.000 }
gfCNCPoint5[6713] = {X 180.8254, Y 35.4572, Z -6.3333, A 0.000, B 0.000, C 0.000 }
gfCNCPoint5[6714] = {X 180.9306, Y 36.0762, Z -6.3333, A 0.000, B 0.000, C 0.000 }
gfCNCPoint5[6715] = {X 181.2237, Y 36.6316, Z -6.3333, A 0.000, B 0.000, C 0.000 }
gfCNCPoint5[6716] = {X 181.6754, Y 37.0677, Z -6.3333, A 0.000, B 0.000, C 0.000 }
gfCNCPoint5[6717] = {X 182.3240, Y 37.4385, Z -6.3333, A 0.000, B 0.000, C 0.000 }
gfCNCPoint5[6718] = {X 183.0176, Y 37.7161, Z -6.3333, A 0.000, B 0.000, C 0.000 }
gfCNCPoint5[6719] = {X 184.4569, Y 38.0378, Z -6.3333, A 0.000, B 0.000, C 0.000 }
gfCNCPoint5[6720] = {X 185.9269, Y 38.1567, Z -6.3333, A 0.000, B 0.000, C 0.000 }
gfCNCPoint5[6721] = {X 187.3992, Y 38.0706, Z -6.3333, A 0.000, B 0.000, C 0.000 }
gfCNCPoint5[6722] = {X 188.8453, Y 37.7811, Z -6.3333, A 0.000, B 0.000, C 0.000 }
gfCNCPoint5[6723] = {X 190.2374, Y 37.2939, Z -6.3333, A 0.000, B 0.000, C 0.000 }
gfCNCPoint5[6724] = {X 191.4936, Y 36.6781, Z -6.3333, A 0.000, B 0.000, C 0.000 }
gfCNCPoint5[6725] = {X 192.6827, Y 35.9410, Z -6.3333, A 0.000, B 0.000, C 0.000 }
gfCNCPoint5[6726] = {X 192.7625, Y 35.1970, Z -6.3333, A 0.000, B 0.000, C 0.000 }
gfCNCPoint5[6727] = {X 192.9744, Y 34.4794, Z -6.3333, A 0.000, B 0.000, C 0.000 }
gfCNCPoint5[6728] = {X 193.3113, Y 33.8113, Z -6.3333, A 0.000, B 0.000, C 0.000 }
gfCNCPoint5[6729] = {X 192.6982, Y 33.9566, Z -6.3333, A 0.000, B 0.000, C 0.000 }
gfCNCPoint5[6730] = {X 190.9622, Y 34.2315, Z -6.3333, A 0.000, B 0.000, C 0.000 }
gfCNCPoint5[6731] = {X 189.2131, Y 34.4053, Z -6.3333, A 0.000, B 0.000, C 0.000 }
gfCNCPoint5[6732] = {X 186.9480, Y 34.5444, Z -6.3333, A 0.000, B 0.000, C 0.000 }
gfCNCPoint5[6733] = {X 182.9921, Y 35.1365, Z -6.3333, A 0.000, B 0.000, C 0.000 }
gfCNCPoint5[6734] = {X 190.9418, Y 34.5683, Z -6.3333, A 0.000, B 0.000, C 0.000 }
gfCNCPoint5[6735] = {X 186.9431, Y 34.4645, Z -6.3333, A 0.000, B 0.000, C 0.000 }
gfCNCPoint5[6736] = {X 182.5509, Y 34.7342, Z -6.3333, A 0.000, B 0.000, C 0.000 }
gfCNCPoint5[6737] = {X 181.6730, Y 34.8409, Z -6.3333, A 0.000, B 0.000, C 0.000 }
gfCNCPoint5[6738] = {X 180.8140, Y 35.0513, Z -6.3333, A 0.000, B 0.000, C 0.000 }
gfCNCPoint5[6739] = {X 180.7584, Y 35.2517, Z -6.3333, A 0.000, B 0.000, C 0.000 }
gfCNCPoint5[6740] = {X 180.7454, Y 35.4593, Z -6.3333, A 0.000, B 0.000, C 0.000 }
gfCNCPoint5[6741] = {X 180.8552, Y 36.1030, Z -6.3333, A 0.000, B 0.000, C 0.000 }
gfCNCPoint5[6742] = {X 181.1603, Y 36.6804, Z -6.3333, A 0.000, B 0.000, C 0.000 }
gfCNCPoint5[6743] = {X 181.6303, Y 37.1337, Z -6.3333, A 0.000, B 0.000, C 0.000 }
gfCNCPoint5[6744] = {X 182.2892, Y 37.5105, Z -6.3333, A 0.000, B 0.000, C 0.000 }
gfCNCPoint5[6745] = {X 182.9939, Y 37.7926, Z -6.3333, A 0.000, B 0.000, C 0.000 }
gfCNCPoint5[6746] = {X 184.4442, Y 38.1168, Z -6.3333, A 0.000, B 0.000, C 0.000 }
gfCNCPoint5[6747] = {X 185.9255, Y 38.2367, Z -6.3333, A 0.000, B 0.000, C 0.000 }
gfCNCPoint5[6748] = {X 187.4091, Y 38.1500, Z -6.3333, A 0.000, B 0.000, C 0.000 }
gfCNCPoint5[6749] = {X 188.8663, Y 37.8583, Z -6.3333, A 0.000, B 0.000, C 0.000 }
gfCNCPoint5[6750] = {X 190.2690, Y 37.3674, Z -6.3333, A 0.000, B 0.000, C 0.000 }
gfCNCPoint5[6751] = {X 191.5504, Y 36.7380, Z -6.3333, A 0.000, B 0.000, C 0.000 }
gfCNCPoint5[6752] = {X 192.7622, Y 35.9832, Z -6.3333, A 0.000, B 0.000, C 0.000 }
gfCNCPoint5[6753] = {X 192.8358, Y 35.2394, Z -6.3333, A 0.000, B 0.000, C 0.000 }
gfCNCPoint5[6754] = {X 193.0437, Y 34.5215, Z -6.3333, A 0.000, B 0.000, C 0.000 }
gfCNCPoint5[6755] = {X 193.3792, Y 33.8536, Z -6.3333, A 0.000, B 0.000, C 0.000 }
gfCNCPoint5[6756] = {X 193.4223, Y 33.7858, Z -6.3333, A 0.000, B 0.000, C 0.000 }
gfCNCPoint5[6757] = {X 193.4668, Y 33.7190, Z -6.3333, A 0.000, B 0.000, C 0.000 }
gfCNCPoint5[6758] = {X 193.3657, Y 33.7162, Z -6.3333, A 0.000, B 0.000, C 0.000 }
gfCNCPoint5[6759] = {X 192.6816, Y 33.8784, Z -6.3333, A 0.000, B 0.000, C 0.000 }
gfCNCPoint5[6760] = {X 190.9512, Y 34.1522, Z -6.3333, A 0.000, B 0.000, C 0.000 }
gfCNCPoint5[6761] = {X 189.2078, Y 34.3255, Z -6.3333, A 0.000, B 0.000, C 0.000 }
gfCNCPoint5[6762] = {X 186.9431, Y 34.4645, Z -6.3333, A 0.000, B 0.000, C 0.000 }
gfCNCPoint5[6763] = {X 182.9872, Y 35.0567, Z -6.3333, A 0.000, B 0.000, C 0.000 }
gfCNCPoint5[6764] = {X 190.9307, Y 34.1395, Z -6.3333, A 0.000, B 0.000, C 0.000 }
gfCNCPoint5[6765] = {X 186.9382, Y 34.3847, Z -6.3333, A 0.000, B 0.000, C 0.000 }
gfCNCPoint5[6766] = {X 182.5460, Y 34.6543, Z -6.3333, A 0.000, B 0.000, C 0.000 }
gfCNCPoint5[6767] = {X 181.6401, Y 34.7656, Z -6.3333, A 0.000, B 0.000, C 0.000 }
gfCNCPoint5[6768] = {X 180.7544, Y 34.9861, Z -6.3333, A 0.000, B 0.000, C 0.000 }
gfCNCPoint5[6769] = {X 180.6830, Y 35.2187, Z -6.3333, A 0.000, B 0.000, C 0.000 }
gfCNCPoint5[6770] = {X 180.6655, Y 35.4613, Z -6.3333, A 0.000, B 0.000, C 0.000 }
gfCNCPoint5[6771] = {X 180.7798, Y 36.1298, Z -6.3333, A 0.000, B 0.000, C 0.000 }
gfCNCPoint5[6772] = {X 181.0969, Y 36.7292, Z -6.3333, A 0.000, B 0.000, C 0.000 }
gfCNCPoint5[6773] = {X 181.5852, Y 37.1998, Z -6.3333, A 0.000, B 0.000, C 0.000 }
gfCNCPoint5[6774] = {X 182.2545, Y 37.5826, Z -6.3333, A 0.000, B 0.000, C 0.000 }
gfCNCPoint5[6775] = {X 182.9702, Y 37.8690, Z -6.3333, A 0.000, B 0.000, C 0.000 }
gfCNCPoint5[6776] = {X 184.4315, Y 38.1958, Z -6.3333, A 0.000, B 0.000, C 0.000 }
gfCNCPoint5[6777] = {X 185.9241, Y 38.3167, Z -6.3333, A 0.000, B 0.000, C 0.000 }
gfCNCPoint5[6778] = {X 187.4189, Y 38.2294, Z -6.3333, A 0.000, B 0.000, C 0.000 }
gfCNCPoint5[6779] = {X 188.8872, Y 37.9355, Z -6.3333, A 0.000, B 0.000, C 0.000 }
gfCNCPoint5[6780] = {X 190.3006, Y 37.4409, Z -6.3333, A 0.000, B 0.000, C 0.000 }
gfCNCPoint5[6781] = {X 191.6075, Y 36.7978, Z -6.3333, A 0.000, B 0.000, C 0.000 }
gfCNCPoint5[6782] = {X 192.8422, Y 36.0250, Z -6.3333, A 0.000, B 0.000, C 0.000 }
gfCNCPoint5[6783] = {X 192.9290, Y 35.1818, Z -6.3333, A 0.000, B 0.000, C 0.000 }
gfCNCPoint5[6784] = {X 193.1917, Y 34.3757, Z -6.3333, A 0.000, B 0.000, C 0.000 }
gfCNCPoint5[6785] = {X 193.6183, Y 33.6431, Z -6.3333, A 0.000, B 0.000, C 0.000 }
gfCNCPoint5[6786] = {X 193.3575, Y 33.6359, Z -6.3333, A 0.000, B 0.000, C 0.000 }
gfCNCPoint5[6787] = {X 192.6650, Y 33.8001, Z -6.3333, A 0.000, B 0.000, C 0.000 }
gfCNCPoint5[6788] = {X 190.9402, Y 34.0730, Z -6.3333, A 0.000, B 0.000, C 0.000 }
gfCNCPoint5[6789] = {X 189.2026, Y 34.2456, Z -6.3333, A 0.000, B 0.000, C 0.000 }
gfCNCPoint5[6790] = {X 186.9382, Y 34.3847, Z -6.3333, A 0.000, B 0.000, C 0.000 }
gfCNCPoint5[6791] = {X 182.9457, Y 34.6298, Z -6.3333, A 0.000, B 0.000, C 0.000 }
gfCNCPoint5[6792] = {X 182.9457, Y 34.6298, Z -3.3333, A 0.000, B 0.000, C 0.000 }
gfCNCPoint5[6793] = {X 182.9457, Y 34.6298, Z 11.0000, A 0.000, B 0.000, C 0.000 }
gfCNCPoint5[6794] = {X 165.6772, Y 73.8165, Z 11.0000, A 0.000, B 0.000, C 0.000 }
gfCNCPoint5[6795] = {X 165.6772, Y 73.8165, Z -2.5000, A 0.000, B 0.000, C 0.000 }
gfCNCPoint5[6796] = {X 161.3996, Y 78.5670, Z -4.2129, A 0.000, B 0.000, C 0.000 }
gfCNCPoint5[6797] = {X 169.3132, Y 78.5670, Z -6.3333, A 0.000, B 0.000, C 0.000 }
gfCNCPoint5[6798] = {X 169.3132, Y 76.1670, Z -6.3333, A 0.000, B 0.000, C 0.000 }
gfCNCPoint5[6799] = {X 171.8361, Y 76.1670, Z -6.3333, A 0.000, B 0.000, C 0.000 }
gfCNCPoint5[6800] = {X 169.3147, Y 73.3634, Z -6.3333, A 0.000, B 0.000, C 0.000 }
gfCNCPoint5[6801] = {X 166.7903, Y 76.1670, Z -6.3333, A 0.000, B 0.000, C 0.000 }
gfCNCPoint5[6802] = {X 169.3132, Y 76.1670, Z -6.3333, A 0.000, B 0.000, C 0.000 }
gfCNCPoint5[6803] = {X 169.3132, Y 78.5670, Z -6.3333, A 0.000, B 0.000, C 0.000 }
gfCNCPoint5[6804] = {X 177.2224, Y 78.5670, Z -6.3333, A 0.000, B 0.000, C 0.000 }
gfCNCPoint5[6805] = {X 169.3158, Y 69.7756, Z -6.3333, A 0.000, B 0.000, C 0.000 }
gfCNCPoint5[6806] = {X 161.3996, Y 78.5670, Z -6.3333, A 0.000, B 0.000, C 0.000 }
gfCNCPoint5[6807] = {X 169.3132, Y 78.5670, Z -6.3333, A 0.000, B 0.000, C 0.000 }
gfCNCPoint5[6808] = {X 169.3132, Y 74.6470, Z -6.3333, A 0.000, B 0.000, C 0.000 }
gfCNCPoint5[6809] = {X 169.3132, Y 78.6470, Z -6.3333, A 0.000, B 0.000, C 0.000 }
gfCNCPoint5[6810] = {X 177.4019, Y 78.6470, Z -6.3333, A 0.000, B 0.000, C 0.000 }
gfCNCPoint5[6811] = {X 169.3159, Y 69.6560, Z -6.3333, A 0.000, B 0.000, C 0.000 }
gfCNCPoint5[6812] = {X 161.2199, Y 78.6470, Z -6.3333, A 0.000, B 0.000, C 0.000 }
gfCNCPoint5[6813] = {X 169.3132, Y 78.6470, Z -6.3333, A 0.000, B 0.000, C 0.000 }
gfCNCPoint5[6814] = {X 169.3132, Y 74.6470, Z -6.3333, A 0.000, B 0.000, C 0.000 }
gfCNCPoint5[6815] = {X 169.3132, Y 74.7270, Z -6.3333, A 0.000, B 0.000, C 0.000 }
gfCNCPoint5[6816] = {X 169.3132, Y 78.7270, Z -6.3333, A 0.000, B 0.000, C 0.000 }
gfCNCPoint5[6817] = {X 177.5814, Y 78.7270, Z -6.3333, A 0.000, B 0.000, C 0.000 }
gfCNCPoint5[6818] = {X 169.3159, Y 69.5364, Z -6.3333, A 0.000, B 0.000, C 0.000 }
gfCNCPoint5[6819] = {X 161.0403, Y 78.7270, Z -6.3333, A 0.000, B 0.000, C 0.000 }
gfCNCPoint5[6820] = {X 169.3132, Y 78.7270, Z -6.3333, A 0.000, B 0.000, C 0.000 }
gfCNCPoint5[6821] = {X 169.3132, Y 74.7270, Z -6.3333, A 0.000, B 0.000, C 0.000 }
gfCNCPoint5[6822] = {X 169.3132, Y 74.8070, Z -6.3333, A 0.000, B 0.000, C 0.000 }
gfCNCPoint5[6823] = {X 169.3132, Y 78.8070, Z -6.3333, A 0.000, B 0.000, C 0.000 }
gfCNCPoint5[6824] = {X 177.7610, Y 78.8070, Z -6.3333, A 0.000, B 0.000, C 0.000 }
gfCNCPoint5[6825] = {X 169.3159, Y 69.4168, Z -6.3333, A 0.000, B 0.000, C 0.000 }
gfCNCPoint5[6826] = {X 160.8606, Y 78.8070, Z -6.3333, A 0.000, B 0.000, C 0.000 }
gfCNCPoint5[6827] = {X 169.3132, Y 78.8070, Z -6.3333, A 0.000, B 0.000, C 0.000 }
gfCNCPoint5[6828] = {X 169.3132, Y 74.8070, Z -6.3333, A 0.000, B 0.000, C 0.000 }
gfCNCPoint5[6829] = {X 169.3132, Y 74.8870, Z -6.3333, A 0.000, B 0.000, C 0.000 }
gfCNCPoint5[6830] = {X 169.3132, Y 78.8870, Z -6.3333, A 0.000, B 0.000, C 0.000 }
gfCNCPoint5[6831] = {X 177.9405, Y 78.8870, Z -6.3333, A 0.000, B 0.000, C 0.000 }
gfCNCPoint5[6832] = {X 169.3160, Y 69.2972, Z -6.3333, A 0.000, B 0.000, C 0.000 }
gfCNCPoint5[6833] = {X 160.6809, Y 78.8870, Z -6.3333, A 0.000, B 0.000, C 0.000 }
gfCNCPoint5[6834] = {X 169.3132, Y 78.8870, Z -6.3333, A 0.000, B 0.000, C 0.000 }
gfCNCPoint5[6835] = {X 169.3132, Y 74.8870, Z -6.3333, A 0.000, B 0.000, C 0.000 }
gfCNCPoint5[6836] = {X 169.3132, Y 74.9670, Z -6.3333, A 0.000, B 0.000, C 0.000 }
gfCNCPoint5[6837] = {X 169.3132, Y 78.9670, Z -6.3333, A 0.000, B 0.000, C 0.000 }
gfCNCPoint5[6838] = {X 178.1201, Y 78.9670, Z -6.3333, A 0.000, B 0.000, C 0.000 }
gfCNCPoint5[6839] = {X 169.3160, Y 69.1776, Z -6.3333, A 0.000, B 0.000, C 0.000 }
gfCNCPoint5[6840] = {X 160.5012, Y 78.9670, Z -6.3333, A 0.000, B 0.000, C 0.000 }
gfCNCPoint5[6841] = {X 169.3132, Y 78.9670, Z -6.3333, A 0.000, B 0.000, C 0.000 }
gfCNCPoint5[6842] = {X 169.3132, Y 74.9670, Z -6.3333, A 0.000, B 0.000, C 0.000 }
gfCNCPoint5[6843] = {X 169.3132, Y 74.9670, Z -3.3333, A 0.000, B 0.000, C 0.000 }
gfCNCPoint5[6844] = {X 169.3132, Y 74.9670, Z 11.0000, A 0.000, B 0.000, C 0.000 }
gfCNCPoint5[6845] = {X 11.7086, Y 37.8762, Z 11.0000, A 0.000, B 0.000, C 0.000 }
gfCNCPoint5[6846] = {X 11.7086, Y 37.8762, Z -2.5000, A 0.000, B 0.000, C 0.000 }
gfCNCPoint5[6847] = {X 12.5124, Y 37.9485, Z -2.7162, A 0.000, B 0.000, C 0.000 }
gfCNCPoint5[6848] = {X 14.1638, Y 37.8337, Z -3.1598, A 0.000, B 0.000, C 0.000 }
gfCNCPoint5[6849] = {X 15.7761, Y 37.4589, Z -3.6033, A 0.000, B 0.000, C 0.000 }
gfCNCPoint5[6850] = {X 16.5088, Y 37.1630, Z -3.8151, A 0.000, B 0.000, C 0.000 }
gfCNCPoint5[6851] = {X 17.3399, Y 36.8273, Z -4.0552, A 0.000, B 0.000, C 0.000 }
gfCNCPoint5[6852] = {X 18.2938, Y 36.3172, Z -4.3451, A 0.000, B 0.000, C 0.000 }
gfCNCPoint5[6853] = {X 19.0345, Y 35.8123, Z -4.5853, A 0.000, B 0.000, C 0.000 }
gfCNCPoint5[6854] = {X 19.0577, Y 35.2981, Z -4.7232, A 0.000, B 0.000, C 0.000 }
gfCNCPoint5[6855] = {X 19.2188, Y 34.6359, Z -4.9058, A 0.000, B 0.000, C 0.000 }
gfCNCPoint5[6856] = {X 19.4343, Y 34.1685, Z -5.0437, A 0.000, B 0.000, C 0.000 }
gfCNCPoint5[6857] = {X 18.2023, Y 34.4168, Z -5.3805, A 0.000, B 0.000, C 0.000 }
gfCNCPoint5[6858] = {X 17.3642, Y 34.5307, Z -5.6071, A 0.000, B 0.000, C 0.000 }
gfCNCPoint5[6859] = {X 16.1106, Y 34.6202, Z -5.9439, A 0.000, B 0.000, C 0.000 }
gfCNCPoint5[6860] = {X 15.3859, Y 34.6740, Z -6.1386, A 0.000, B 0.000, C 0.000 }
gfCNCPoint5[6861] = {X 14.6608, Y 34.7236, Z -6.3333, A 0.000, B 0.000, C 0.000 }
gfCNCPoint5[6862] = {X 12.2607, Y 34.8762, Z -6.3333, A 0.000, B 0.000, C 0.000 }
gfCNCPoint5[6863] = {X 9.8591, Y 35.0059, Z -6.3333, A 0.000, B 0.000, C 0.000 }
gfCNCPoint5[6864] = {X 8.7539, Y 35.0958, Z -6.3333, A 0.000, B 0.000, C 0.000 }
gfCNCPoint5[6865] = {X 7.6658, Y 35.3097, Z -6.3333, A 0.000, B 0.000, C 0.000 }
gfCNCPoint5[6866] = {X 7.6562, Y 35.3713, Z -6.3333, A 0.000, B 0.000, C 0.000 }
gfCNCPoint5[6867] = {X 7.6529, Y 35.4335, Z -6.3333, A 0.000, B 0.000, C 0.000 }
gfCNCPoint5[6868] = {X 7.7535, Y 36.0259, Z -6.3333, A 0.000, B 0.000, C 0.000 }
gfCNCPoint5[6869] = {X 8.0477, Y 36.5498, Z -6.3333, A 0.000, B 0.000, C 0.000 }
gfCNCPoint5[6870] = {X 8.5011, Y 36.9440, Z -6.3333, A 0.000, B 0.000, C 0.000 }
gfCNCPoint5[6871] = {X 9.2742, Y 37.3361, Z -6.3333, A 0.000, B 0.000, C 0.000 }
gfCNCPoint5[6872] = {X 10.0972, Y 37.6086, Z -6.3333, A 0.000, B 0.000, C 0.000 }
gfCNCPoint5[6873] = {X 11.3815, Y 37.8452, Z -6.3333, A 0.000, B 0.000, C 0.000 }
gfCNCPoint5[6874] = {X 12.6854, Y 37.9188, Z -6.3333, A 0.000, B 0.000, C 0.000 }
gfCNCPoint5[6875] = {X 13.9883, Y 37.8282, Z -6.3333, A 0.000, B 0.000, C 0.000 }
gfCNCPoint5[6876] = {X 15.2695, Y 37.5750, Z -6.3333, A 0.000, B 0.000, C 0.000 }
gfCNCPoint5[6877] = {X 16.5088, Y 37.1630, Z -6.3333, A 0.000, B 0.000, C 0.000 }
gfCNCPoint5[6878] = {X 17.8079, Y 36.5554, Z -6.3333, A 0.000, B 0.000, C 0.000 }
gfCNCPoint5[6879] = {X 19.0345, Y 35.8123, Z -6.3333, A 0.000, B 0.000, C 0.000 }
gfCNCPoint5[6880] = {X 19.1547, Y 34.9710, Z -6.3333, A 0.000, B 0.000, C 0.000 }
gfCNCPoint5[6881] = {X 19.4343, Y 34.1685, Z -6.3333, A 0.000, B 0.000, C 0.000 }
gfCNCPoint5[6882] = {X 17.7797, Y 34.4474, Z -6.3333, A 0.000, B 0.000, C 0.000 }
gfCNCPoint5[6883] = {X 16.1106, Y 34.6202, Z -6.3333, A 0.000, B 0.000, C 0.000 }
gfCNCPoint5[6884] = {X 15.3858, Y 34.6729, Z -6.3333, A 0.000, B 0.000, C 0.000 }
gfCNCPoint5[6885] = {X 14.6608, Y 34.7236, Z -6.3333, A 0.000, B 0.000, C 0.000 }
gfCNCPoint5[6886] = {X 18.6546, Y 34.7197, Z -6.3333, A 0.000, B 0.000, C 0.000 }
gfCNCPoint5[6887] = {X 14.6554, Y 34.6438, Z -6.3333, A 0.000, B 0.000, C 0.000 }
gfCNCPoint5[6888] = {X 12.2589, Y 34.7962, Z -6.3333, A 0.000, B 0.000, C 0.000 }
gfCNCPoint5[6889] = {X 9.8610, Y 34.9258, Z -6.3333, A 0.000, B 0.000, C 0.000 }
gfCNCPoint5[6890] = {X 8.7211, Y 35.0197, Z -6.3333, A 0.000, B 0.000, C 0.000 }
gfCNCPoint5[6891] = {X 7.5995, Y 35.2442, Z -6.3333, A 0.000, B 0.000, C 0.000 }
gfCNCPoint5[6892] = {X 7.5797, Y 35.3378, Z -6.3333, A 0.000, B 0.000, C 0.000 }
gfCNCPoint5[6893] = {X 7.5729, Y 35.4333, Z -6.3333, A 0.000, B 0.000, C 0.000 }
gfCNCPoint5[6894] = {X 7.6781, Y 36.0526, Z -6.3333, A 0.000, B 0.000, C 0.000 }
gfCNCPoint5[6895] = {X 7.9857, Y 36.6003, Z -6.3333, A 0.000, B 0.000, C 0.000 }
gfCNCPoint5[6896] = {X 8.4597, Y 37.0125, Z -6.3333, A 0.000, B 0.000, C 0.000 }
gfCNCPoint5[6897] = {X 9.2435, Y 37.4099, Z -6.3333, A 0.000, B 0.000, C 0.000 }
gfCNCPoint5[6898] = {X 10.0778, Y 37.6862, Z -6.3333, A 0.000, B 0.000, C 0.000 }
gfCNCPoint5[6899] = {X 11.3720, Y 37.9246, Z -6.3333, A 0.000, B 0.000, C 0.000 }
gfCNCPoint5[6900] = {X 12.6860, Y 37.9988, Z -6.3333, A 0.000, B 0.000, C 0.000 }
gfCNCPoint5[6901] = {X 13.9988, Y 37.9075, Z -6.3333, A 0.000, B 0.000, C 0.000 }
gfCNCPoint5[6902] = {X 15.2899, Y 37.6523, Z -6.3333, A 0.000, B 0.000, C 0.000 }
gfCNCPoint5[6903] = {X 16.5387, Y 37.2372, Z -6.3333, A 0.000, B 0.000, C 0.000 }
gfCNCPoint5[6904] = {X 17.8633, Y 36.6165, Z -6.3333, A 0.000, B 0.000, C 0.000 }
gfCNCPoint5[6905] = {X 19.1128, Y 35.8556, Z -6.3333, A 0.000, B 0.000, C 0.000 }
gfCNCPoint5[6906] = {X 19.2470, Y 34.9314, Z -6.3333, A 0.000, B 0.000, C 0.000 }
gfCNCPoint5[6907] = {X 19.5768, Y 34.0576, Z -6.3333, A 0.000, B 0.000, C 0.000 }
gfCNCPoint5[6908] = {X 17.8489, Y 34.3571, Z -6.3333, A 0.000, B 0.000, C 0.000 }
gfCNCPoint5[6909] = {X 16.1048, Y 34.5404, Z -6.3333, A 0.000, B 0.000, C 0.000 }
gfCNCPoint5[6910] = {X 15.3802, Y 34.5931, Z -6.3333, A 0.000, B 0.000, C 0.000 }
gfCNCPoint5[6911] = {X 14.6554, Y 34.6438, Z -6.3333, A 0.000, B 0.000, C 0.000 }
gfCNCPoint5[6912] = {X 10.7037, Y 35.2634, Z -6.3333, A 0.000, B 0.000, C 0.000 }
gfCNCPoint5[6913] = {X 18.6492, Y 34.6399, Z -6.3333, A 0.000, B 0.000, C 0.000 }
gfCNCPoint5[6914] = {X 14.6499, Y 34.5639, Z -6.3333, A 0.000, B 0.000, C 0.000 }
gfCNCPoint5[6915] = {X 12.2547, Y 34.7163, Z -6.3333, A 0.000, B 0.000, C 0.000 }
gfCNCPoint5[6916] = {X 9.8581, Y 34.8458, Z -6.3333, A 0.000, B 0.000, C 0.000 }
gfCNCPoint5[6917] = {X 8.6875, Y 34.9436, Z -6.3333, A 0.000, B 0.000, C 0.000 }
gfCNCPoint5[6918] = {X 7.5365, Y 35.1781, Z -6.3333, A 0.000, B 0.000, C 0.000 }
gfCNCPoint5[6919] = {X 7.5041, Y 35.3037, Z -6.3333, A 0.000, B 0.000, C 0.000 }
gfCNCPoint5[6920] = {X 7.4929, Y 35.4330, Z -6.3333, A 0.000, B 0.000, C 0.000 }
gfCNCPoint5[6921] = {X 7.6027, Y 36.0792, Z -6.3333, A 0.000, B 0.000, C 0.000 }
gfCNCPoint5[6922] = {X 7.9236, Y 36.6508, Z -6.3333, A 0.000, B 0.000, C 0.000 }
gfCNCPoint5[6923] = {X 8.4183, Y 37.0809, Z -6.3333, A 0.000, B 0.000, C 0.000 }
gfCNCPoint5[6924] = {X 9.2127, Y 37.4838, Z -6.3333, A 0.000, B 0.000, C 0.000 }
gfCNCPoint5[6925] = {X 10.0584, Y 37.7638, Z -6.3333, A 0.000, B 0.000, C 0.000 }
gfCNCPoint5[6926] = {X 11.3625, Y 38.0040, Z -6.3333, A 0.000, B 0.000, C 0.000 }
gfCNCPoint5[6927] = {X 12.6865, Y 38.0788, Z -6.3333, A 0.000, B 0.000, C 0.000 }
gfCNCPoint5[6928] = {X 14.0094, Y 37.9868, Z -6.3333, A 0.000, B 0.000, C 0.000 }
gfCNCPoint5[6929] = {X 15.3103, Y 37.7297, Z -6.3333, A 0.000, B 0.000, C 0.000 }
gfCNCPoint5[6930] = {X 16.5687, Y 37.3114, Z -6.3333, A 0.000, B 0.000, C 0.000 }
gfCNCPoint5[6931] = {X 17.9191, Y 36.6773, Z -6.3333, A 0.000, B 0.000, C 0.000 }
gfCNCPoint5[6932] = {X 19.1915, Y 35.8986, Z -6.3333, A 0.000, B 0.000, C 0.000 }
gfCNCPoint5[6933] = {X 19.2642, Y 35.2210, Z -6.3333, A 0.000, B 0.000, C 0.000 }
gfCNCPoint5[6934] = {X 19.4446, Y 34.5637, Z -6.3333, A 0.000, B 0.000, C 0.000 }
gfCNCPoint5[6935] = {X 19.7280, Y 33.9439, Z -6.3333, A 0.000, B 0.000, C 0.000 }
gfCNCPoint5[6936] = {X 17.9226, Y 34.2660, Z -6.3333, A 0.000, B 0.000, C 0.000 }
gfCNCPoint5[6937] = {X 16.0990, Y 34.4607, Z -6.3333, A 0.000, B 0.000, C 0.000 }
gfCNCPoint5[6938] = {X 15.3745, Y 34.5133, Z -6.3333, A 0.000, B 0.000, C 0.000 }
gfCNCPoint5[6939] = {X 14.6499, Y 34.5639, Z -6.3333, A 0.000, B 0.000, C 0.000 }
gfCNCPoint5[6940] = {X 10.6982, Y 35.1836, Z -6.3333, A 0.000, B 0.000, C 0.000 }
gfCNCPoint5[6941] = {X 18.6437, Y 34.5601, Z -6.3333, A 0.000, B 0.000, C 0.000 }
gfCNCPoint5[6942] = {X 14.6444, Y 34.4841, Z -6.3333, A 0.000, B 0.000, C 0.000 }
gfCNCPoint5[6943] = {X 12.2505, Y 34.6364, Z -6.3333, A 0.000, B 0.000, C 0.000 }
gfCNCPoint5[6944] = {X 9.8551, Y 34.7659, Z -6.3333, A 0.000, B 0.000, C 0.000 }
gfCNCPoint5[6945] = {X 8.6553, Y 34.8674, Z -6.3333, A 0.000, B 0.000, C 0.000 }
gfCNCPoint5[6946] = {X 7.4762, Y 35.1114, Z -6.3333, A 0.000, B 0.000, C 0.000 }
gfCNCPoint5[6947] = {X 7.4291, Y 35.2690, Z -6.3333, A 0.000, B 0.000, C 0.000 }
gfCNCPoint5[6948] = {X 7.4129, Y 35.4327, Z -6.3333, A 0.000, B 0.000, C 0.000 }
gfCNCPoint5[6949] = {X 7.5272, Y 36.1059, Z -6.3333, A 0.000, B 0.000, C 0.000 }
gfCNCPoint5[6950] = {X 7.8616, Y 36.7013, Z -6.3333, A 0.000, B 0.000, C 0.000 }
gfCNCPoint5[6951] = {X 8.3769, Y 37.1494, Z -6.3333, A 0.000, B 0.000, C 0.000 }
gfCNCPoint5[6952] = {X 9.1820, Y 37.5576, Z -6.3333, A 0.000, B 0.000, C 0.000 }
gfCNCPoint5[6953] = {X 10.0389, Y 37.8414, Z -6.3333, A 0.000, B 0.000, C 0.000 }
gfCNCPoint5[6954] = {X 11.3530, Y 38.0835, Z -6.3333, A 0.000, B 0.000, C 0.000 }
gfCNCPoint5[6955] = {X 12.6870, Y 38.1588, Z -6.3333, A 0.000, B 0.000, C 0.000 }
gfCNCPoint5[6956] = {X 14.0199, Y 38.0661, Z -6.3333, A 0.000, B 0.000, C 0.000 }
gfCNCPoint5[6957] = {X 15.3307, Y 37.8070, Z -6.3333, A 0.000, B 0.000, C 0.000 }
gfCNCPoint5[6958] = {X 16.5986, Y 37.3855, Z -6.3333, A 0.000, B 0.000, C 0.000 }
gfCNCPoint5[6959] = {X 17.9750, Y 36.7381, Z -6.3333, A 0.000, B 0.000, C 0.000 }
gfCNCPoint5[6960] = {X 19.2706, Y 35.9411, Z -6.3333, A 0.000, B 0.000, C 0.000 }
gfCNCPoint5[6961] = {X 19.3492, Y 35.2030, Z -6.3333, A 0.000, B 0.000, C 0.000 }
gfCNCPoint5[6962] = {X 19.5577, Y 34.4907, Z -6.3333, A 0.000, B 0.000, C 0.000 }
gfCNCPoint5[6963] = {X 19.8896, Y 33.8267, Z -6.3333, A 0.000, B 0.000, C 0.000 }
gfCNCPoint5[6964] = {X 18.0016, Y 34.1737, Z -6.3333, A 0.000, B 0.000, C 0.000 }
gfCNCPoint5[6965] = {X 16.0932, Y 34.3809, Z -6.3333, A 0.000, B 0.000, C 0.000 }
gfCNCPoint5[6966] = {X 15.3689, Y 34.4335, Z -6.3333, A 0.000, B 0.000, C 0.000 }
gfCNCPoint5[6967] = {X 14.6444, Y 34.4841, Z -6.3333, A 0.000, B 0.000, C 0.000 }
gfCNCPoint5[6968] = {X 10.6927, Y 35.1038, Z -6.3333, A 0.000, B 0.000, C 0.000 }
gfCNCPoint5[6969] = {X 18.6383, Y 34.4803, Z -6.3333, A 0.000, B 0.000, C 0.000 }
gfCNCPoint5[6970] = {X 14.6390, Y 34.4043, Z -6.3333, A 0.000, B 0.000, C 0.000 }
gfCNCPoint5[6971] = {X 12.2463, Y 34.5565, Z -6.3333, A 0.000, B 0.000, C 0.000 }
gfCNCPoint5[6972] = {X 9.8522, Y 34.6859, Z -6.3333, A 0.000, B 0.000, C 0.000 }
gfCNCPoint5[6973] = {X 8.6242, Y 34.7911, Z -6.3333, A 0.000, B 0.000, C 0.000 }
gfCNCPoint5[6974] = {X 7.4180, Y 35.0443, Z -6.3333, A 0.000, B 0.000, C 0.000 }
gfCNCPoint5[6975] = {X 7.3548, Y 35.2339, Z -6.3333, A 0.000, B 0.000, C 0.000 }
gfCNCPoint5[6976] = {X 7.3329, Y 35.4324, Z -6.3333, A 0.000, B 0.000, C 0.000 }
gfCNCPoint5[6977] = {X 7.3996, Y 35.9620, Z -6.3333, A 0.000, B 0.000, C 0.000 }
gfCNCPoint5[6978] = {X 7.5990, Y 36.4572, Z -6.3333, A 0.000, B 0.000, C 0.000 }
gfCNCPoint5[6979] = {X 7.9180, Y 36.8852, Z -6.3333, A 0.000, B 0.000, C 0.000 }
gfCNCPoint5[6980] = {X 8.3355, Y 37.2178, Z -6.3333, A 0.000, B 0.000, C 0.000 }
gfCNCPoint5[6981] = {X 9.1512, Y 37.6315, Z -6.3333, A 0.000, B 0.000, C 0.000 }
gfCNCPoint5[6982] = {X 10.0195, Y 37.9190, Z -6.3333, A 0.000, B 0.000, C 0.000 }
gfCNCPoint5[6983] = {X 11.3435, Y 38.1629, Z -6.3333, A 0.000, B 0.000, C 0.000 }
gfCNCPoint5[6984] = {X 12.6875, Y 38.2388, Z -6.3333, A 0.000, B 0.000, C 0.000 }
gfCNCPoint5[6985] = {X 14.0305, Y 38.1454, Z -6.3333, A 0.000, B 0.000, C 0.000 }
gfCNCPoint5[6986] = {X 15.3511, Y 37.8844, Z -6.3333, A 0.000, B 0.000, C 0.000 }
gfCNCPoint5[6987] = {X 16.6286, Y 37.4597, Z -6.3333, A 0.000, B 0.000, C 0.000 }
gfCNCPoint5[6988] = {X 18.0312, Y 36.7986, Z -6.3333, A 0.000, B 0.000, C 0.000 }
gfCNCPoint5[6989] = {X 19.3501, Y 35.9832, Z -6.3333, A 0.000, B 0.000, C 0.000 }
gfCNCPoint5[6990] = {X 19.4352, Y 35.1815, Z -6.3333, A 0.000, B 0.000, C 0.000 }
gfCNCPoint5[6991] = {X 19.6763, Y 34.4122, Z -6.3333, A 0.000, B 0.000, C 0.000 }
gfCNCPoint5[6992] = {X 20.0640, Y 33.7053, Z -6.3333, A 0.000, B 0.000, C 0.000 }
gfCNCPoint5[6993] = {X 18.0872, Y 34.0802, Z -6.3333, A 0.000, B 0.000, C 0.000 }
gfCNCPoint5[6994] = {X 16.0874, Y 34.3011, Z -6.3333, A 0.000, B 0.000, C 0.000 }
gfCNCPoint5[6995] = {X 15.3633, Y 34.3537, Z -6.3333, A 0.000, B 0.000, C 0.000 }
gfCNCPoint5[6996] = {X 14.6390, Y 34.4043, Z -6.3333, A 0.000, B 0.000, C 0.000 }
gfCNCPoint5[6997] = {X 10.6873, Y 35.0240, Z -6.3333, A 0.000, B 0.000, C 0.000 }
gfCNCPoint5[6998] = {X 14.7700, Y 36.3198, Z -6.3333, A 0.000, B 0.000, C 0.000 }
gfCNCPoint5[6999] = {X 14.6335, Y 34.3245, Z -6.3333, A 0.000, B 0.000, C 0.000 }
gfCNCPoint5[7000] = {X 12.2420, Y 34.4766, Z -6.3333, A 0.000, B 0.000, C 0.000 }
gfCNCPoint5[7001] = {X 9.8492, Y 34.6060, Z -6.3333, A 0.000, B 0.000, C 0.000 }
gfCNCPoint5[7002] = {X 8.5940, Y 34.7147, Z -6.3333, A 0.000, B 0.000, C 0.000 }
gfCNCPoint5[7003] = {X 7.3616, Y 34.9769, Z -6.3333, A 0.000, B 0.000, C 0.000 }
gfCNCPoint5[7004] = {X 7.2808, Y 35.1982, Z -6.3333, A 0.000, B 0.000, C 0.000 }
gfCNCPoint5[7005] = {X 7.2529, Y 35.4322, Z -6.3333, A 0.000, B 0.000, C 0.000 }
gfCNCPoint5[7006] = {X 7.3222, Y 35.9821, Z -6.3333, A 0.000, B 0.000, C 0.000 }
gfCNCPoint5[7007] = {X 7.5293, Y 36.4963, Z -6.3333, A 0.000, B 0.000, C 0.000 }
gfCNCPoint5[7008] = {X 7.8605, Y 36.9408, Z -6.3333, A 0.000, B 0.000, C 0.000 }
gfCNCPoint5[7009] = {X 8.2940, Y 37.2863, Z -6.3333, A 0.000, B 0.000, C 0.000 }
gfCNCPoint5[7010] = {X 9.1205, Y 37.7053, Z -6.3333, A 0.000, B 0.000, C 0.000 }
gfCNCPoint5[7011] = {X 10.0001, Y 37.9966, Z -6.3333, A 0.000, B 0.000, C 0.000 }
gfCNCPoint5[7012] = {X 11.3339, Y 38.2423, Z -6.3333, A 0.000, B 0.000, C 0.000 }
gfCNCPoint5[7013] = {X 12.6880, Y 38.3188, Z -6.3333, A 0.000, B 0.000, C 0.000 }
gfCNCPoint5[7014] = {X 14.0410, Y 38.2247, Z -6.3333, A 0.000, B 0.000, C 0.000 }
gfCNCPoint5[7015] = {X 15.3715, Y 37.9617, Z -6.3333, A 0.000, B 0.000, C 0.000 }
gfCNCPoint5[7016] = {X 16.6585, Y 37.5339, Z -6.3333, A 0.000, B 0.000, C 0.000 }
gfCNCPoint5[7017] = {X 18.0876, Y 36.8590, Z -6.3333, A 0.000, B 0.000, C 0.000 }
gfCNCPoint5[7018] = {X 19.4300, Y 36.0248, Z -6.3333, A 0.000, B 0.000, C 0.000 }
gfCNCPoint5[7019] = {X 19.5226, Y 35.1553, Z -6.3333, A 0.000, B 0.000, C 0.000 }
gfCNCPoint5[7020] = {X 19.8019, Y 34.3266, Z -6.3333, A 0.000, B 0.000, C 0.000 }
gfCNCPoint5[7021] = {X 20.2547, Y 33.5784, Z -6.3333, A 0.000, B 0.000, C 0.000 }
gfCNCPoint5[7022] = {X 18.1812, Y 33.9850, Z -6.3333, A 0.000, B 0.000, C 0.000 }
gfCNCPoint5[7023] = {X 16.0816, Y 34.2213, Z -6.3333, A 0.000, B 0.000, C 0.000 }
gfCNCPoint5[7024] = {X 15.3576, Y 34.2739, Z -6.3333, A 0.000, B 0.000, C 0.000 }
gfCNCPoint5[7025] = {X 14.6335, Y 34.3245, Z -6.3333, A 0.000, B 0.000, C 0.000 }
gfCNCPoint5[7026] = {X 14.7700, Y 36.3198, Z -6.3333, A 0.000, B 0.000, C 0.000 }
gfCNCPoint5[7027] = {X 14.7700, Y 36.3198, Z -3.3333, A 0.000, B 0.000, C 0.000 }
gfCNCPoint5[7028] = {X 14.7700, Y 36.3198, Z 11.0000, A 0.000, B 0.000, C 0.000 }
gfCNCPoint5[7029] = {X 15.0775, Y 19.4935, Z 11.0000, A 0.000, B 0.000, C 0.000 }
gfCNCPoint5[7030] = {X 15.0775, Y 19.4935, Z -2.5000, A 0.000, B 0.000, C 0.000 }
gfCNCPoint5[7031] = {X 14.5040, Y 19.3637, Z -2.6575, A 0.000, B 0.000, C 0.000 }
gfCNCPoint5[7032] = {X 13.3045, Y 19.2501, Z -2.9804, A 0.000, B 0.000, C 0.000 }
gfCNCPoint5[7033] = {X 12.0998, Y 19.2675, Z -3.3032, A 0.000, B 0.000, C 0.000 }
gfCNCPoint5[7034] = {X 11.2937, Y 19.3831, Z -3.5214, A 0.000, B 0.000, C 0.000 }
gfCNCPoint5[7035] = {X 10.6069, Y 19.4911, Z -3.7077, A 0.000, B 0.000, C 0.000 }
gfCNCPoint5[7036] = {X 9.8992, Y 19.6140, Z -3.9002, A 0.000, B 0.000, C 0.000 }
gfCNCPoint5[7037] = {X 8.6146, Y 20.0604, Z -4.2646, A 0.000, B 0.000, C 0.000 }
gfCNCPoint5[7038] = {X 7.9832, Y 20.4028, Z -4.4570, A 0.000, B 0.000, C 0.000 }
gfCNCPoint5[7039] = {X 7.9271, Y 20.9144, Z -4.5950, A 0.000, B 0.000, C 0.000 }
gfCNCPoint5[7040] = {X 7.4477, Y 22.1349, Z -4.9463, A 0.000, B 0.000, C 0.000 }
gfCNCPoint5[7041] = {X 7.1407, Y 22.5480, Z -5.0842, A 0.000, B 0.000, C 0.000 }
gfCNCPoint5[7042] = {X 8.7362, Y 22.3428, Z -5.5152, A 0.000, B 0.000, C 0.000 }
gfCNCPoint5[7043] = {X 9.6128, Y 22.2722, Z -5.7509, A 0.000, B 0.000, C 0.000 }
gfCNCPoint5[7044] = {X 11.2206, Y 22.2193, Z -6.1819, A 0.000, B 0.000, C 0.000 }
gfCNCPoint5[7045] = {X 11.5030, Y 22.2094, Z -6.2576, A 0.000, B 0.000, C 0.000 }
gfCNCPoint5[7046] = {X 11.7853, Y 22.1981, Z -6.3333, A 0.000, B 0.000, C 0.000 }
gfCNCPoint5[7047] = {X 14.1121, Y 22.0787, Z -6.3333, A 0.000, B 0.000, C 0.000 }
gfCNCPoint5[7048] = {X 16.4356, Y 21.9080, Z -6.3333, A 0.000, B 0.000, C 0.000 }
gfCNCPoint5[7049] = {X 17.0513, Y 21.8311, Z -6.3333, A 0.000, B 0.000, C 0.000 }
gfCNCPoint5[7050] = {X 17.6520, Y 21.6762, Z -6.3333, A 0.000, B 0.000, C 0.000 }
gfCNCPoint5[7051] = {X 17.6738, Y 21.2170, Z -6.3333, A 0.000, B 0.000, C 0.000 }
gfCNCPoint5[7052] = {X 17.5243, Y 20.7824, Z -6.3333, A 0.000, B 0.000, C 0.000 }
gfCNCPoint5[7053] = {X 17.2245, Y 20.4339, Z -6.3333, A 0.000, B 0.000, C 0.000 }
gfCNCPoint5[7054] = {X 16.3055, Y 19.8933, Z -6.3333, A 0.000, B 0.000, C 0.000 }
gfCNCPoint5[7055] = {X 15.2983, Y 19.5435, Z -6.3333, A 0.000, B 0.000, C 0.000 }
gfCNCPoint5[7056] = {X 13.9732, Y 19.3273, Z -6.3333, A 0.000, B 0.000, C 0.000 }
gfCNCPoint5[7057] = {X 12.6318, Y 19.2736, Z -6.3333, A 0.000, B 0.000, C 0.000 }
gfCNCPoint5[7058] = {X 11.2937, Y 19.3831, Z -6.3333, A 0.000, B 0.000, C 0.000 }
gfCNCPoint5[7059] = {X 10.6069, Y 19.4911, Z -6.3333, A 0.000, B 0.000, C 0.000 }
gfCNCPoint5[7060] = {X 9.2579, Y 19.8401, Z -6.3333, A 0.000, B 0.000, C 0.000 }
gfCNCPoint5[7061] = {X 7.9832, Y 20.4028, Z -6.3333, A 0.000, B 0.000, C 0.000 }
gfCNCPoint5[7062] = {X 7.8308, Y 21.1640, Z -6.3333, A 0.000, B 0.000, C 0.000 }
gfCNCPoint5[7063] = {X 7.5470, Y 21.8865, Z -6.3333, A 0.000, B 0.000, C 0.000 }
gfCNCPoint5[7064] = {X 7.1407, Y 22.5480, Z -6.3333, A 0.000, B 0.000, C 0.000 }
gfCNCPoint5[7065] = {X 9.1768, Y 22.3352, Z -6.3333, A 0.000, B 0.000, C 0.000 }
gfCNCPoint5[7066] = {X 11.2206, Y 22.2193, Z -6.3333, A 0.000, B 0.000, C 0.000 }
gfCNCPoint5[7067] = {X 11.5030, Y 22.2090, Z -6.3333, A 0.000, B 0.000, C 0.000 }
gfCNCPoint5[7068] = {X 11.7853, Y 22.1981, Z -6.3333, A 0.000, B 0.000, C 0.000 }
gfCNCPoint5[7069] = {X 7.7929, Y 22.0899, Z -6.3333, A 0.000, B 0.000, C 0.000 }
gfCNCPoint5[7070] = {X 11.7885, Y 22.2780, Z -6.3333, A 0.000, B 0.000, C 0.000 }
gfCNCPoint5[7071] = {X 14.1142, Y 22.1587, Z -6.3333, A 0.000, B 0.000, C 0.000 }
gfCNCPoint5[7072] = {X 16.4366, Y 21.9881, Z -6.3333, A 0.000, B 0.000, C 0.000 }
gfCNCPoint5[7073] = {X 17.0859, Y 21.9059, Z -6.3333, A 0.000, B 0.000, C 0.000 }
gfCNCPoint5[7074] = {X 17.7185, Y 21.7384, Z -6.3333, A 0.000, B 0.000, C 0.000 }
gfCNCPoint5[7075] = {X 17.7568, Y 21.2348, Z -6.3333, A 0.000, B 0.000, C 0.000 }
gfCNCPoint5[7076] = {X 17.6005, Y 20.7546, Z -6.3333, A 0.000, B 0.000, C 0.000 }
gfCNCPoint5[7077] = {X 17.2730, Y 20.3702, Z -6.3333, A 0.000, B 0.000, C 0.000 }
gfCNCPoint5[7078] = {X 16.3395, Y 19.8210, Z -6.3333, A 0.000, B 0.000, C 0.000 }
gfCNCPoint5[7079] = {X 15.3164, Y 19.4656, Z -6.3333, A 0.000, B 0.000, C 0.000 }
gfCNCPoint5[7080] = {X 13.9815, Y 19.2477, Z -6.3333, A 0.000, B 0.000, C 0.000 }
gfCNCPoint5[7081] = {X 12.6299, Y 19.1936, Z -6.3333, A 0.000, B 0.000, C 0.000 }
gfCNCPoint5[7082] = {X 11.2818, Y 19.3040, Z -6.3333, A 0.000, B 0.000, C 0.000 }
gfCNCPoint5[7083] = {X 10.5939, Y 19.4122, Z -6.3333, A 0.000, B 0.000, C 0.000 }
gfCNCPoint5[7084] = {X 9.2121, Y 19.7714, Z -6.3333, A 0.000, B 0.000, C 0.000 }
gfCNCPoint5[7085] = {X 7.9080, Y 20.3527, Z -6.3333, A 0.000, B 0.000, C 0.000 }
gfCNCPoint5[7086] = {X 7.7436, Y 21.1765, Z -6.3333, A 0.000, B 0.000, C 0.000 }
gfCNCPoint5[7087] = {X 7.4228, Y 21.9529, Z -6.3333, A 0.000, B 0.000, C 0.000 }
gfCNCPoint5[7088] = {X 6.9579, Y 22.6526, Z -6.3333, A 0.000, B 0.000, C 0.000 }
gfCNCPoint5[7089] = {X 9.0862, Y 22.4228, Z -6.3333, A 0.000, B 0.000, C 0.000 }
gfCNCPoint5[7090] = {X 11.2233, Y 22.2992, Z -6.3333, A 0.000, B 0.000, C 0.000 }
gfCNCPoint5[7091] = {X 11.5059, Y 22.2890, Z -6.3333, A 0.000, B 0.000, C 0.000 }
gfCNCPoint5[7092] = {X 11.7885, Y 22.2780, Z -6.3333, A 0.000, B 0.000, C 0.000 }
gfCNCPoint5[7093] = {X 15.7560, Y 21.7694, Z -6.3333, A 0.000, B 0.000, C 0.000 }
gfCNCPoint5[7094] = {X 7.7962, Y 22.1699, Z -6.3333, A 0.000, B 0.000, C 0.000 }
gfCNCPoint5[7095] = {X 11.7917, Y 22.3579, Z -6.3333, A 0.000, B 0.000, C 0.000 }
gfCNCPoint5[7096] = {X 14.1187, Y 22.2386, Z -6.3333, A 0.000, B 0.000, C 0.000 }
gfCNCPoint5[7097] = {X 16.4424, Y 22.0679, Z -6.3333, A 0.000, B 0.000, C 0.000 }
gfCNCPoint5[7098] = {X 17.1221, Y 21.9803, Z -6.3333, A 0.000, B 0.000, C 0.000 }
gfCNCPoint5[7099] = {X 17.7835, Y 21.8007, Z -6.3333, A 0.000, B 0.000, C 0.000 }
gfCNCPoint5[7100] = {X 17.8393, Y 21.2530, Z -6.3333, A 0.000, B 0.000, C 0.000 }
gfCNCPoint5[7101] = {X 17.6767, Y 20.7271, Z -6.3333, A 0.000, B 0.000, C 0.000 }
gfCNCPoint5[7102] = {X 17.3214, Y 20.3065, Z -6.3333, A 0.000, B 0.000, C 0.000 }
gfCNCPoint5[7103] = {X 16.3736, Y 19.7486, Z -6.3333, A 0.000, B 0.000, C 0.000 }
gfCNCPoint5[7104] = {X 15.3346, Y 19.3876, Z -6.3333, A 0.000, B 0.000, C 0.000 }
gfCNCPoint5[7105] = {X 13.9897, Y 19.1681, Z -6.3333, A 0.000, B 0.000, C 0.000 }
gfCNCPoint5[7106] = {X 12.6281, Y 19.1136, Z -6.3333, A 0.000, B 0.000, C 0.000 }
gfCNCPoint5[7107] = {X 11.2699, Y 19.2249, Z -6.3333, A 0.000, B 0.000, C 0.000 }
gfCNCPoint5[7108] = {X 10.5808, Y 19.3332, Z -6.3333, A 0.000, B 0.000, C 0.000 }
gfCNCPoint5[7109] = {X 9.6302, Y 19.5534, Z -6.3333, A 0.000, B 0.000, C 0.000 }
gfCNCPoint5[7110] = {X 8.7100, Y 19.8782, Z -6.3333, A 0.000, B 0.000, C 0.000 }
gfCNCPoint5[7111] = {X 7.8318, Y 20.3034, Z -6.3333, A 0.000, B 0.000, C 0.000 }
gfCNCPoint5[7112] = {X 7.8284, Y 20.3447, Z -6.3333, A 0.000, B 0.000, C 0.000 }
gfCNCPoint5[7113] = {X 7.6463, Y 21.2195, Z -6.3333, A 0.000, B 0.000, C 0.000 }
gfCNCPoint5[7114] = {X 7.2850, Y 22.0367, Z -6.3333, A 0.000, B 0.000, C 0.000 }
gfCNCPoint5[7115] = {X 6.7604, Y 22.7601, Z -6.3333, A 0.000, B 0.000, C 0.000 }
gfCNCPoint5[7116] = {X 8.9883, Y 22.5114, Z -6.3333, A 0.000, B 0.000, C 0.000 }
gfCNCPoint5[7117] = {X 11.2260, Y 22.3792, Z -6.3333, A 0.000, B 0.000, C 0.000 }
gfCNCPoint5[7118] = {X 11.5089, Y 22.3689, Z -6.3333, A 0.000, B 0.000, C 0.000 }
gfCNCPoint5[7119] = {X 11.7917, Y 22.3579, Z -6.3333, A 0.000, B 0.000, C 0.000 }
gfCNCPoint5[7120] = {X 15.7593, Y 21.8493, Z -6.3333, A 0.000, B 0.000, C 0.000 }
gfCNCPoint5[7121] = {X 7.7994, Y 22.2498, Z -6.3333, A 0.000, B 0.000, C 0.000 }
gfCNCPoint5[7122] = {X 11.7949, Y 22.4379, Z -6.3333, A 0.000, B 0.000, C 0.000 }
gfCNCPoint5[7123] = {X 14.1231, Y 22.3184, Z -6.3333, A 0.000, B 0.000, C 0.000 }
gfCNCPoint5[7124] = {X 16.4481, Y 22.1477, Z -6.3333, A 0.000, B 0.000, C 0.000 }
gfCNCPoint5[7125] = {X 17.1577, Y 22.0547, Z -6.3333, A 0.000, B 0.000, C 0.000 }
gfCNCPoint5[7126] = {X 17.8473, Y 21.8631, Z -6.3333, A 0.000, B 0.000, C 0.000 }
gfCNCPoint5[7127] = {X 17.9257, Y 21.4215, Z -6.3333, A 0.000, B 0.000, C 0.000 }
gfCNCPoint5[7128] = {X 17.8665, Y 20.9769, Z -6.3333, A 0.000, B 0.000, C 0.000 }
gfCNCPoint5[7129] = {X 17.6752, Y 20.5713, Z -6.3333, A 0.000, B 0.000, C 0.000 }
gfCNCPoint5[7130] = {X 17.3698, Y 20.2428, Z -6.3333, A 0.000, B 0.000, C 0.000 }
gfCNCPoint5[7131] = {X 16.4076, Y 19.6762, Z -6.3333, A 0.000, B 0.000, C 0.000 }
gfCNCPoint5[7132] = {X 15.3528, Y 19.3097, Z -6.3333, A 0.000, B 0.000, C 0.000 }
gfCNCPoint5[7133] = {X 13.9979, Y 19.0886, Z -6.3333, A 0.000, B 0.000, C 0.000 }
gfCNCPoint5[7134] = {X 12.6262, Y 19.0337, Z -6.3333, A 0.000, B 0.000, C 0.000 }
gfCNCPoint5[7135] = {X 11.2580, Y 19.1458, Z -6.3333, A 0.000, B 0.000, C 0.000 }
gfCNCPoint5[7136] = {X 10.5678, Y 19.2543, Z -6.3333, A 0.000, B 0.000, C 0.000 }
gfCNCPoint5[7137] = {X 9.5945, Y 19.4805, Z -6.3333, A 0.000, B 0.000, C 0.000 }
gfCNCPoint5[7138] = {X 8.6530, Y 19.8153, Z -6.3333, A 0.000, B 0.000, C 0.000 }
gfCNCPoint5[7139] = {X 7.7554, Y 20.2544, Z -6.3333, A 0.000, B 0.000, C 0.000 }
gfCNCPoint5[7140] = {X 7.7492, Y 20.3325, Z -6.3333, A 0.000, B 0.000, C 0.000 }
gfCNCPoint5[7141] = {X 7.5473, Y 21.2643, Z -6.3333, A 0.000, B 0.000, C 0.000 }
gfCNCPoint5[7142] = {X 7.1385, Y 22.1257, Z -6.3333, A 0.000, B 0.000, C 0.000 }
gfCNCPoint5[7143] = {X 6.5443, Y 22.8713, Z -6.3333, A 0.000, B 0.000, C 0.000 }
gfCNCPoint5[7144] = {X 8.8809, Y 22.6010, Z -6.3333, A 0.000, B 0.000, C 0.000 }
gfCNCPoint5[7145] = {X 11.2288, Y 22.4591, Z -6.3333, A 0.000, B 0.000, C 0.000 }
gfCNCPoint5[7146] = {X 11.5119, Y 22.4489, Z -6.3333, A 0.000, B 0.000, C 0.000 }
gfCNCPoint5[7147] = {X 11.7949, Y 22.4379, Z -6.3333, A 0.000, B 0.000, C 0.000 }
gfCNCPoint5[7148] = {X 15.7625, Y 21.9293, Z -6.3333, A 0.000, B 0.000, C 0.000 }
gfCNCPoint5[7149] = {X 7.8026, Y 22.3297, Z -6.3333, A 0.000, B 0.000, C 0.000 }
gfCNCPoint5[7150] = {X 11.7982, Y 22.5178, Z -6.3333, A 0.000, B 0.000, C 0.000 }
gfCNCPoint5[7151] = {X 14.1276, Y 22.3983, Z -6.3333, A 0.000, B 0.000, C 0.000 }
gfCNCPoint5[7152] = {X 16.4539, Y 22.2275, Z -6.3333, A 0.000, B 0.000, C 0.000 }
gfCNCPoint5[7153] = {X 17.1928, Y 22.1292, Z -6.3333, A 0.000, B 0.000, C 0.000 }
gfCNCPoint5[7154] = {X 17.9099, Y 21.9256, Z -6.3333, A 0.000, B 0.000, C 0.000 }
gfCNCPoint5[7155] = {X 18.0048, Y 21.4520, Z -6.3333, A 0.000, B 0.000, C 0.000 }
gfCNCPoint5[7156] = {X 17.9484, Y 20.9722, Z -6.3333, A 0.000, B 0.000, C 0.000 }
gfCNCPoint5[7157] = {X 17.7463, Y 20.5336, Z -6.3333, A 0.000, B 0.000, C 0.000 }
gfCNCPoint5[7158] = {X 17.4182, Y 20.1791, Z -6.3333, A 0.000, B 0.000, C 0.000 }
gfCNCPoint5[7159] = {X 16.4416, Y 19.6037, Z -6.3333, A 0.000, B 0.000, C 0.000 }
gfCNCPoint5[7160] = {X 15.3709, Y 19.2318, Z -6.3333, A 0.000, B 0.000, C 0.000 }
gfCNCPoint5[7161] = {X 14.0061, Y 19.0090, Z -6.3333, A 0.000, B 0.000, C 0.000 }
gfCNCPoint5[7162] = {X 12.6243, Y 18.9537, Z -6.3333, A 0.000, B 0.000, C 0.000 }
gfCNCPoint5[7163] = {X 11.2461, Y 19.0667, Z -6.3333, A 0.000, B 0.000, C 0.000 }
gfCNCPoint5[7164] = {X 10.5547, Y 19.1754, Z -6.3333, A 0.000, B 0.000, C 0.000 }
gfCNCPoint5[7165] = {X 9.5587, Y 19.4076, Z -6.3333, A 0.000, B 0.000, C 0.000 }
gfCNCPoint5[7166] = {X 8.5959, Y 19.7526, Z -6.3333, A 0.000, B 0.000, C 0.000 }
gfCNCPoint5[7167] = {X 7.6791, Y 20.2056, Z -6.3333, A 0.000, B 0.000, C 0.000 }
gfCNCPoint5[7168] = {X 7.6695, Y 20.3254, Z -6.3333, A 0.000, B 0.000, C 0.000 }
gfCNCPoint5[7169] = {X 7.5231, Y 21.0761, Z -6.3333, A 0.000, B 0.000, C 0.000 }
gfCNCPoint5[7170] = {X 7.2391, Y 21.7863, Z -6.3333, A 0.000, B 0.000, C 0.000 }
gfCNCPoint5[7171] = {X 6.8276, Y 22.4310, Z -6.3333, A 0.000, B 0.000, C 0.000 }
gfCNCPoint5[7172] = {X 6.3030, Y 22.9876, Z -6.3333, A 0.000, B 0.000, C 0.000 }
gfCNCPoint5[7173] = {X 8.7607, Y 22.6920, Z -6.3333, A 0.000, B 0.000, C 0.000 }
gfCNCPoint5[7174] = {X 11.2315, Y 22.5391, Z -6.3333, A 0.000, B 0.000, C 0.000 }
gfCNCPoint5[7175] = {X 11.5148, Y 22.5288, Z -6.3333, A 0.000, B 0.000, C 0.000 }
gfCNCPoint5[7176] = {X 11.7982, Y 22.5178, Z -6.3333, A 0.000, B 0.000, C 0.000 }
gfCNCPoint5[7177] = {X 15.7657, Y 22.0092, Z -6.3333, A 0.000, B 0.000, C 0.000 }
gfCNCPoint5[7178] = {X 11.7264, Y 22.6007, Z -6.3333, A 0.000, B 0.000, C 0.000 }
gfCNCPoint5[7179] = {X 11.8014, Y 22.5977, Z -6.3333, A 0.000, B 0.000, C 0.000 }
gfCNCPoint5[7180] = {X 14.1321, Y 22.4782, Z -6.3333, A 0.000, B 0.000, C 0.000 }
gfCNCPoint5[7181] = {X 16.4597, Y 22.3073, Z -6.3333, A 0.000, B 0.000, C 0.000 }
gfCNCPoint5[7182] = {X 17.2274, Y 22.2037, Z -6.3333, A 0.000, B 0.000, C 0.000 }
gfCNCPoint5[7183] = {X 17.9716, Y 21.9881, Z -6.3333, A 0.000, B 0.000, C 0.000 }
gfCNCPoint5[7184] = {X 18.0834, Y 21.4827, Z -6.3333, A 0.000, B 0.000, C 0.000 }
gfCNCPoint5[7185] = {X 18.0302, Y 20.9678, Z -6.3333, A 0.000, B 0.000, C 0.000 }
gfCNCPoint5[7186] = {X 17.8173, Y 20.4960, Z -6.3333, A 0.000, B 0.000, C 0.000 }
gfCNCPoint5[7187] = {X 17.4665, Y 20.1153, Z -6.3333, A 0.000, B 0.000, C 0.000 }
gfCNCPoint5[7188] = {X 16.4756, Y 19.5313, Z -6.3333, A 0.000, B 0.000, C 0.000 }
gfCNCPoint5[7189] = {X 15.3891, Y 19.1539, Z -6.3333, A 0.000, B 0.000, C 0.000 }
gfCNCPoint5[7190] = {X 14.0143, Y 18.9294, Z -6.3333, A 0.000, B 0.000, C 0.000 }
gfCNCPoint5[7191] = {X 12.6225, Y 18.8737, Z -6.3333, A 0.000, B 0.000, C 0.000 }
gfCNCPoint5[7192] = {X 11.2342, Y 18.9876, Z -6.3333, A 0.000, B 0.000, C 0.000 }
gfCNCPoint5[7193] = {X 10.5417, Y 19.0964, Z -6.3333, A 0.000, B 0.000, C 0.000 }
gfCNCPoint5[7194] = {X 9.5230, Y 19.3348, Z -6.3333, A 0.000, B 0.000, C 0.000 }
gfCNCPoint5[7195] = {X 8.5388, Y 19.6900, Z -6.3333, A 0.000, B 0.000, C 0.000 }
gfCNCPoint5[7196] = {X 7.6027, Y 20.1571, Z -6.3333, A 0.000, B 0.000, C 0.000 }
gfCNCPoint5[7197] = {X 7.5898, Y 20.3183, Z -6.3333, A 0.000, B 0.000, C 0.000 }
gfCNCPoint5[7198] = {X 7.4462, Y 21.0541, Z -6.3333, A 0.000, B 0.000, C 0.000 }
gfCNCPoint5[7199] = {X 7.1678, Y 21.7501, Z -6.3333, A 0.000, B 0.000, C 0.000 }
gfCNCPoint5[7200] = {X 6.7644, Y 22.3820, Z -6.3333, A 0.000, B 0.000, C 0.000 }
gfCNCPoint5[7201] = {X 6.2502, Y 22.9275, Z -6.3333, A 0.000, B 0.000, C 0.000 }
gfCNCPoint5[7202] = {X 6.2082, Y 22.9638, Z -6.3333, A 0.000, B 0.000, C 0.000 }
gfCNCPoint5[7203] = {X 6.1658, Y 22.9996, Z -6.3333, A 0.000, B 0.000, C 0.000 }
gfCNCPoint5[7204] = {X 6.1509, Y 23.0915, Z -6.3333, A 0.000, B 0.000, C 0.000 }
gfCNCPoint5[7205] = {X 6.2329, Y 23.0790, Z -6.3333, A 0.000, B 0.000, C 0.000 }
gfCNCPoint5[7206] = {X 6.3148, Y 23.0667, Z -6.3333, A 0.000, B 0.000, C 0.000 }
gfCNCPoint5[7207] = {X 8.7680, Y 22.7717, Z -6.3333, A 0.000, B 0.000, C 0.000 }
gfCNCPoint5[7208] = {X 11.2342, Y 22.6190, Z -6.3333, A 0.000, B 0.000, C 0.000 }
gfCNCPoint5[7209] = {X 11.5178, Y 22.6088, Z -6.3333, A 0.000, B 0.000, C 0.000 }
gfCNCPoint5[7210] = {X 11.8014, Y 22.5977, Z -6.3333, A 0.000, B 0.000, C 0.000 }
gfCNCPoint5[7211] = {X 11.7209, Y 20.5994, Z -6.3333, A 0.000, B 0.000, C 0.000 }
gfCNCPoint5[7212] = {X 11.7209, Y 20.5994, Z -3.3333, A 0.000, B 0.000, C 0.000 }
gfCNCPoint5[7213] = {X 11.7209, Y 20.5994, Z 11.0000, A 0.000, B 0.000, C 0.000 }
gfCNCPoint5[7214] = {X 15.0786, Y 19.4941, Z 11.0000, A 0.000, B 0.000, C 0.000 }
gfCNCPoint5[7215] = {X 15.0786, Y 19.4941, Z -3.3333, A 0.000, B 0.000, C 0.000 }
gfCNCPoint5[7216] = {X 14.5040, Y 19.3640, Z -3.4912, A 0.000, B 0.000, C 0.000 }
gfCNCPoint5[7217] = {X 13.3045, Y 19.2504, Z -3.8140, A 0.000, B 0.000, C 0.000 }
gfCNCPoint5[7218] = {X 12.0998, Y 19.2678, Z -4.1369, A 0.000, B 0.000, C 0.000 }
gfCNCPoint5[7219] = {X 11.2937, Y 19.3835, Z -4.3551, A 0.000, B 0.000, C 0.000 }
gfCNCPoint5[7220] = {X 10.6069, Y 19.4914, Z -4.5414, A 0.000, B 0.000, C 0.000 }
gfCNCPoint5[7221] = {X 9.8993, Y 19.6143, Z -4.7338, A 0.000, B 0.000, C 0.000 }
gfCNCPoint5[7222] = {X 8.6144, Y 20.0608, Z -5.0983, A 0.000, B 0.000, C 0.000 }
gfCNCPoint5[7223] = {X 7.9831, Y 20.4032, Z -5.2907, A 0.000, B 0.000, C 0.000 }
gfCNCPoint5[7224] = {X 7.9270, Y 20.9148, Z -5.4286, A 0.000, B 0.000, C 0.000 }
gfCNCPoint5[7225] = {X 7.4480, Y 22.1345, Z -5.7797, A 0.000, B 0.000, C 0.000 }
gfCNCPoint5[7226] = {X 7.1410, Y 22.5476, Z -5.9177, A 0.000, B 0.000, C 0.000 }
gfCNCPoint5[7227] = {X 8.7365, Y 22.3425, Z -6.3487, A 0.000, B 0.000, C 0.000 }
gfCNCPoint5[7228] = {X 9.6128, Y 22.2719, Z -6.5843, A 0.000, B 0.000, C 0.000 }
gfCNCPoint5[7229] = {X 11.2206, Y 22.2189, Z -7.0153, A 0.000, B 0.000, C 0.000 }
gfCNCPoint5[7230] = {X 11.5029, Y 22.2091, Z -7.0910, A 0.000, B 0.000, C 0.000 }
gfCNCPoint5[7231] = {X 11.7851, Y 22.1977, Z -7.1667, A 0.000, B 0.000, C 0.000 }
gfCNCPoint5[7232] = {X 14.1117, Y 22.0784, Z -7.1667, A 0.000, B 0.000, C 0.000 }
gfCNCPoint5[7233] = {X 16.4350, Y 21.9080, Z -7.1667, A 0.000, B 0.000, C 0.000 }
gfCNCPoint5[7234] = {X 17.0508, Y 21.8308, Z -7.1667, A 0.000, B 0.000, C 0.000 }
gfCNCPoint5[7235] = {X 17.6517, Y 21.6759, Z -7.1667, A 0.000, B 0.000, C 0.000 }
gfCNCPoint5[7236] = {X 17.6735, Y 21.2170, Z -7.1667, A 0.000, B 0.000, C 0.000 }
gfCNCPoint5[7237] = {X 17.5240, Y 20.7826, Z -7.1667, A 0.000, B 0.000, C 0.000 }
gfCNCPoint5[7238] = {X 17.2245, Y 20.4342, Z -7.1667, A 0.000, B 0.000, C 0.000 }
gfCNCPoint5[7239] = {X 16.3055, Y 19.8936, Z -7.1667, A 0.000, B 0.000, C 0.000 }
gfCNCPoint5[7240] = {X 15.2983, Y 19.5438, Z -7.1667, A 0.000, B 0.000, C 0.000 }
gfCNCPoint5[7241] = {X 13.9732, Y 19.3276, Z -7.1667, A 0.000, B 0.000, C 0.000 }
gfCNCPoint5[7242] = {X 12.6318, Y 19.2739, Z -7.1667, A 0.000, B 0.000, C 0.000 }
gfCNCPoint5[7243] = {X 11.2937, Y 19.3835, Z -7.1667, A 0.000, B 0.000, C 0.000 }
gfCNCPoint5[7244] = {X 10.6069, Y 19.4914, Z -7.1667, A 0.000, B 0.000, C 0.000 }
gfCNCPoint5[7245] = {X 9.2579, Y 19.8404, Z -7.1667, A 0.000, B 0.000, C 0.000 }
gfCNCPoint5[7246] = {X 7.9831, Y 20.4032, Z -7.1667, A 0.000, B 0.000, C 0.000 }
gfCNCPoint5[7247] = {X 7.8308, Y 21.1641, Z -7.1667, A 0.000, B 0.000, C 0.000 }
gfCNCPoint5[7248] = {X 7.5471, Y 21.8864, Z -7.1667, A 0.000, B 0.000, C 0.000 }
gfCNCPoint5[7249] = {X 7.1410, Y 22.5476, Z -7.1667, A 0.000, B 0.000, C 0.000 }
gfCNCPoint5[7250] = {X 9.1769, Y 22.3348, Z -7.1667, A 0.000, B 0.000, C 0.000 }
gfCNCPoint5[7251] = {X 11.2206, Y 22.2189, Z -7.1667, A 0.000, B 0.000, C 0.000 }
gfCNCPoint5[7252] = {X 11.5029, Y 22.2087, Z -7.1667, A 0.000, B 0.000, C 0.000 }
gfCNCPoint5[7253] = {X 11.7851, Y 22.1977, Z -7.1667, A 0.000, B 0.000, C 0.000 }
gfCNCPoint5[7254] = {X 7.7927, Y 22.0898, Z -7.1667, A 0.000, B 0.000, C 0.000 }
